gfCNCPoint1[26395] = {X 109.0469, Y 40.8285, Z -2.1667, A 0.000, B 0.000, C 0.000 }
gfCNCPoint1[26396] = {X 109.0468, Y 39.7004, Z -2.1667, A 0.000, B 0.000, C 0.000 }
gfCNCPoint1[26397] = {X 108.5557, Y 40.9005, Z -2.1667, A 0.000, B 0.000, C 0.000 }
gfCNCPoint1[26398] = {X 108.5557, Y 40.9005, Z 0.8333, A 0.000, B 0.000, C 0.000 }
gfCNCPoint1[26399] = {X 108.5557, Y 40.9005, Z 11.0000, A 0.000, B 0.000, C 0.000 }
gfCNCPoint1[26400] = {X 95.6842, Y 40.8760, Z 11.0000, A 0.000, B 0.000, C 0.000 }
gfCNCPoint1[26401] = {X 95.6842, Y 40.8760, Z 1.6667, A 0.000, B 0.000, C 0.000 }
gfCNCPoint1[26402] = {X 95.6842, Y 40.8760, Z -2.1667, A 0.000, B 0.000, C 0.000 }
gfCNCPoint1[26403] = {X 95.2101, Y 39.7165, Z -2.1667, A 0.000, B 0.000, C 0.000 }
gfCNCPoint1[26404] = {X 95.2102, Y 40.8690, Z -2.1667, A 0.000, B 0.000, C 0.000 }
gfCNCPoint1[26405] = {X 95.7335, Y 41.4123, Z -2.1667, A 0.000, B 0.000, C 0.000 }
gfCNCPoint1[26406] = {X 96.1583, Y 42.0355, Z -2.1667, A 0.000, B 0.000, C 0.000 }
gfCNCPoint1[26407] = {X 95.6842, Y 40.8760, Z -2.1667, A 0.000, B 0.000, C 0.000 }
gfCNCPoint1[26408] = {X 95.6842, Y 40.8760, Z 0.8333, A 0.000, B 0.000, C 0.000 }
gfCNCPoint1[26409] = {X 95.6842, Y 40.8760, Z 11.0000, A 0.000, B 0.000, C 0.000 }
gfCNCPoint1[26410] = {X -7.6965, Y 43.1560, Z 11.0000, A 0.000, B 0.000, C 0.000 }
gfCNCPoint1[26411] = {X -7.6965, Y 43.1560, Z 0.8333, A 0.000, B 0.000, C 0.000 }
gfCNCPoint1[26412] = {X -7.6965, Y 43.1560, Z -2.1667, A 0.000, B 0.000, C 0.000 }
gfCNCPoint1[26413] = {X -3.6965, Y 30.8015, Z -2.1667, A 0.000, B 0.000, C 0.000 }
gfCNCPoint1[26414] = {X -3.3664, Y 29.8871, Z -2.1667, A 0.000, B 0.000, C 0.000 }
gfCNCPoint1[26415] = {X -2.9760, Y 28.9968, Z -2.1667, A 0.000, B 0.000, C 0.000 }
gfCNCPoint1[26416] = {X -2.3495, Y 27.8703, Z -2.1667, A 0.000, B 0.000, C 0.000 }
gfCNCPoint1[26417] = {X -1.5931, Y 26.8265, Z -2.1667, A 0.000, B 0.000, C 0.000 }
gfCNCPoint1[26418] = {X -0.7177, Y 25.8802, Z -2.1667, A 0.000, B 0.000, C 0.000 }
gfCNCPoint1[26419] = {X 0.2642, Y 25.0451, Z -2.1667, A 0.000, B 0.000, C 0.000 }
gfCNCPoint1[26420] = {X 1.3386, Y 24.3329, Z -2.1667, A 0.000, B 0.000, C 0.000 }
gfCNCPoint1[26421] = {X 0.5787, Y 23.9225, Z -2.1667, A 0.000, B 0.000, C 0.000 }
gfCNCPoint1[26422] = {X -0.0865, Y 23.3717, Z -2.1667, A 0.000, B 0.000, C 0.000 }
gfCNCPoint1[26423] = {X -0.6312, Y 22.7015, Z -2.1667, A 0.000, B 0.000, C 0.000 }
gfCNCPoint1[26424] = {X -1.0345, Y 21.9378, Z -2.1667, A 0.000, B 0.000, C 0.000 }
gfCNCPoint1[26425] = {X -3.6458, Y 15.5423, Z -2.1667, A 0.000, B 0.000, C 0.000 }
gfCNCPoint1[26426] = {X -3.6716, Y 15.4775, Z -2.1667, A 0.000, B 0.000, C 0.000 }
gfCNCPoint1[26427] = {X -3.6965, Y 15.4122, Z -2.1667, A 0.000, B 0.000, C 0.000 }
gfCNCPoint1[26428] = {X -7.6965, Y 4.6517, Z -2.1667, A 0.000, B 0.000, C 0.000 }
gfCNCPoint1[26429] = {X -7.6965, Y 4.6517, Z 0.8333, A 0.000, B 0.000, C 0.000 }
gfCNCPoint1[26430] = {X -7.6965, Y 4.6517, Z 11.0000, A 0.000, B 0.000, C 0.000 }
gfCNCPoint1[26431] = {X -7.6965, Y 16.4123, Z 11.0000, A 0.000, B 0.000, C 0.000 }
gfCNCPoint1[26432] = {X -7.6965, Y 16.4123, Z 0.8333, A 0.000, B 0.000, C 0.000 }
gfCNCPoint1[26433] = {X -7.6965, Y 16.4123, Z -2.1667, A 0.000, B 0.000, C 0.000 }
gfCNCPoint1[26434] = {X -4.8869, Y 16.4123, Z -2.1667, A 0.000, B 0.000, C 0.000 }
gfCNCPoint1[26435] = {X -3.6965, Y 12.5935, Z -2.1667, A 0.000, B 0.000, C 0.000 }
gfCNCPoint1[26436] = {X -3.6605, Y 12.4832, Z -2.1667, A 0.000, B 0.000, C 0.000 }
gfCNCPoint1[26437] = {X -3.6215, Y 12.3739, Z -2.1667, A 0.000, B 0.000, C 0.000 }
gfCNCPoint1[26438] = {X -3.1666, Y 11.4827, Z -2.1667, A 0.000, B 0.000, C 0.000 }
gfCNCPoint1[26439] = {X -2.5188, Y 10.7200, Z -2.1667, A 0.000, B 0.000, C 0.000 }
gfCNCPoint1[26440] = {X -1.7129, Y 10.1268, Z -2.1667, A 0.000, B 0.000, C 0.000 }
gfCNCPoint1[26441] = {X -1.1157, Y 9.7861, Z -2.1667, A 0.000, B 0.000, C 0.000 }
gfCNCPoint1[26442] = {X -0.2291, Y 9.4045, Z -2.1667, A 0.000, B 0.000, C 0.000 }
gfCNCPoint1[26443] = {X 0.7202, Y 9.2292, Z -2.1667, A 0.000, B 0.000, C 0.000 }
gfCNCPoint1[26444] = {X 1.6847, Y 9.2691, Z -2.1667, A 0.000, B 0.000, C 0.000 }
gfCNCPoint1[26445] = {X 2.6162, Y 9.5222, Z -2.1667, A 0.000, B 0.000, C 0.000 }
gfCNCPoint1[26446] = {X 3.3958, Y 9.1594, Z -2.1667, A 0.000, B 0.000, C 0.000 }
gfCNCPoint1[26447] = {X 4.1961, Y 8.8448, Z -2.1667, A 0.000, B 0.000, C 0.000 }
gfCNCPoint1[26448] = {X 6.1070, Y 8.1762, Z -2.1667, A 0.000, B 0.000, C 0.000 }
gfCNCPoint1[26449] = {X 8.0685, Y 7.6747, Z -2.1667, A 0.000, B 0.000, C 0.000 }
gfCNCPoint1[26450] = {X 10.0658, Y 7.3442, Z -2.1667, A 0.000, B 0.000, C 0.000 }
gfCNCPoint1[26451] = {X 12.0843, Y 7.1871, Z -2.1667, A 0.000, B 0.000, C 0.000 }
gfCNCPoint1[26452] = {X 14.1088, Y 7.2045, Z -2.1667, A 0.000, B 0.000, C 0.000 }
gfCNCPoint1[26453] = {X 16.1242, Y 7.3964, Z -2.1667, A 0.000, B 0.000, C 0.000 }
gfCNCPoint1[26454] = {X 17.9474, Y 7.7301, Z -2.1667, A 0.000, B 0.000, C 0.000 }
gfCNCPoint1[26455] = {X 19.7250, Y 8.2552, Z -2.1667, A 0.000, B 0.000, C 0.000 }
gfCNCPoint1[26456] = {X 21.4368, Y 8.9658, Z -2.1667, A 0.000, B 0.000, C 0.000 }
gfCNCPoint1[26457] = {X 23.0637, Y 9.8538, Z -2.1667, A 0.000, B 0.000, C 0.000 }
gfCNCPoint1[26458] = {X 24.5873, Y 10.9093, Z -2.1667, A 0.000, B 0.000, C 0.000 }
gfCNCPoint1[26459] = {X 25.6719, Y 11.8584, Z -2.1667, A 0.000, B 0.000, C 0.000 }
gfCNCPoint1[26460] = {X 26.6450, Y 12.9216, Z -2.1667, A 0.000, B 0.000, C 0.000 }
gfCNCPoint1[26461] = {X 27.4945, Y 14.0858, Z -2.1667, A 0.000, B 0.000, C 0.000 }
gfCNCPoint1[26462] = {X 28.2102, Y 15.3368, Z -2.1667, A 0.000, B 0.000, C 0.000 }
gfCNCPoint1[26463] = {X 28.7831, Y 16.6592, Z -2.1667, A 0.000, B 0.000, C 0.000 }
gfCNCPoint1[26464] = {X 29.2588, Y 18.3155, Z -2.1667, A 0.000, B 0.000, C 0.000 }
gfCNCPoint1[26465] = {X 29.5409, Y 20.0155, Z -2.1667, A 0.000, B 0.000, C 0.000 }
gfCNCPoint1[26466] = {X 29.6260, Y 21.7366, Z -2.1667, A 0.000, B 0.000, C 0.000 }
gfCNCPoint1[26467] = {X 29.5127, Y 23.4561, Z -2.1667, A 0.000, B 0.000, C 0.000 }
gfCNCPoint1[26468] = {X 29.2026, Y 25.1512, Z -2.1667, A 0.000, B 0.000, C 0.000 }
gfCNCPoint1[26469] = {X 28.7606, Y 26.5973, Z -2.1667, A 0.000, B 0.000, C 0.000 }
gfCNCPoint1[26470] = {X 28.1355, Y 27.9743, Z -2.1667, A 0.000, B 0.000, C 0.000 }
gfCNCPoint1[26471] = {X 27.3378, Y 29.2590, Z -2.1667, A 0.000, B 0.000, C 0.000 }
gfCNCPoint1[26472] = {X 26.3810, Y 30.4299, Z -2.1667, A 0.000, B 0.000, C 0.000 }
gfCNCPoint1[26473] = {X 25.2809, Y 31.4676, Z -2.1667, A 0.000, B 0.000, C 0.000 }
gfCNCPoint1[26474] = {X 26.0850, Y 31.8097, Z -2.1667, A 0.000, B 0.000, C 0.000 }
gfCNCPoint1[26475] = {X 26.8038, Y 32.3066, Z -2.1667, A 0.000, B 0.000, C 0.000 }
gfCNCPoint1[26476] = {X 27.4079, Y 32.9381, Z -2.1667, A 0.000, B 0.000, C 0.000 }
gfCNCPoint1[26477] = {X 27.8726, Y 33.6781, Z -2.1667, A 0.000, B 0.000, C 0.000 }
gfCNCPoint1[26478] = {X 30.9100, Y 39.9530, Z -2.1667, A 0.000, B 0.000, C 0.000 }
gfCNCPoint1[26479] = {X 31.2306, Y 40.8622, Z -2.1667, A 0.000, B 0.000, C 0.000 }
gfCNCPoint1[26480] = {X 31.3415, Y 41.8197, Z -2.1667, A 0.000, B 0.000, C 0.000 }
gfCNCPoint1[26481] = {X 31.2374, Y 42.7781, Z -2.1667, A 0.000, B 0.000, C 0.000 }
gfCNCPoint1[26482] = {X 30.9234, Y 43.6895, Z -2.1667, A 0.000, B 0.000, C 0.000 }
gfCNCPoint1[26483] = {X 30.4150, Y 44.5085, Z -2.1667, A 0.000, B 0.000, C 0.000 }
gfCNCPoint1[26484] = {X 29.7377, Y 45.1945, Z -2.1667, A 0.000, B 0.000, C 0.000 }
gfCNCPoint1[26485] = {X 29.2014, Y 45.6281, Z -2.1667, A 0.000, B 0.000, C 0.000 }
gfCNCPoint1[26486] = {X 28.4966, Y 46.0912, Z -2.1667, A 0.000, B 0.000, C 0.000 }
gfCNCPoint1[26487] = {X 27.7155, Y 46.4091, Z -2.1667, A 0.000, B 0.000, C 0.000 }
gfCNCPoint1[26488] = {X 26.8877, Y 46.5699, Z -2.1667, A 0.000, B 0.000, C 0.000 }
gfCNCPoint1[26489] = {X 26.0445, Y 46.5675, Z -2.1667, A 0.000, B 0.000, C 0.000 }
gfCNCPoint1[26490] = {X 25.2176, Y 46.4020, Z -2.1667, A 0.000, B 0.000, C 0.000 }
gfCNCPoint1[26491] = {X 23.1996, Y 47.4597, Z -2.1667, A 0.000, B 0.000, C 0.000 }
gfCNCPoint1[26492] = {X 21.1036, Y 48.3530, Z -2.1667, A 0.000, B 0.000, C 0.000 }
gfCNCPoint1[26493] = {X 18.9430, Y 49.0760, Z -2.1667, A 0.000, B 0.000, C 0.000 }
gfCNCPoint1[26494] = {X 16.8434, Y 49.5947, Z -2.1667, A 0.000, B 0.000, C 0.000 }
gfCNCPoint1[26495] = {X 14.7038, Y 49.9107, Z -2.1667, A 0.000, B 0.000, C 0.000 }
gfCNCPoint1[26496] = {X 12.5438, Y 50.0209, Z -2.1667, A 0.000, B 0.000, C 0.000 }
gfCNCPoint1[26497] = {X 10.3832, Y 49.9245, Z -2.1667, A 0.000, B 0.000, C 0.000 }
gfCNCPoint1[26498] = {X 8.2417, Y 49.6223, Z -2.1667, A 0.000, B 0.000, C 0.000 }
gfCNCPoint1[26499] = {X 6.4092, Y 49.1801, Z -2.1667, A 0.000, B 0.000, C 0.000 }
gfCNCPoint1[26500] = {X 4.6364, Y 48.5391, Z -2.1667, A 0.000, B 0.000, C 0.000 }
gfCNCPoint1[26501] = {X 2.9448, Y 47.7071, Z -2.1667, A 0.000, B 0.000, C 0.000 }
gfCNCPoint1[26502] = {X 1.3550, Y 46.6941, Z -2.1667, A 0.000, B 0.000, C 0.000 }
gfCNCPoint1[26503] = {X 0.0296, Y 45.6271, Z -2.1667, A 0.000, B 0.000, C 0.000 }
gfCNCPoint1[26504] = {X -1.1487, Y 44.3994, Z -2.1667, A 0.000, B 0.000, C 0.000 }
gfCNCPoint1[26505] = {X -2.1603, Y 43.0312, Z -2.1667, A 0.000, B 0.000, C 0.000 }
gfCNCPoint1[26506] = {X -2.9888, Y 41.5449, Z -2.1667, A 0.000, B 0.000, C 0.000 }
gfCNCPoint1[26507] = {X -3.6205, Y 39.9650, Z -2.1667, A 0.000, B 0.000, C 0.000 }
gfCNCPoint1[26508] = {X -3.6590, Y 39.8451, Z -2.1667, A 0.000, B 0.000, C 0.000 }
gfCNCPoint1[26509] = {X -3.6965, Y 39.7249, Z -2.1667, A 0.000, B 0.000, C 0.000 }
gfCNCPoint1[26510] = {X -4.8683, Y 35.9004, Z -2.1667, A 0.000, B 0.000, C 0.000 }
gfCNCPoint1[26511] = {X -7.9903, Y 36.0269, Z -2.1667, A 0.000, B 0.000, C 0.000 }
gfCNCPoint1[26512] = {X -7.9903, Y 36.0269, Z 0.8333, A 0.000, B 0.000, C 0.000 }
gfCNCPoint1[26513] = {X -7.9903, Y 36.0269, Z 11.0000, A 0.000, B 0.000, C 0.000 }
gfCNCPoint1[26514] = {X 608.0000, Y 40.1203, Z 11.0000, A 0.000, B 0.000, C 0.000 }
gfCNCPoint1[26515] = {X 608.0000, Y 40.1203, Z 0.8333, A 0.000, B 0.000, C 0.000 }
gfCNCPoint1[26516] = {X 608.0000, Y 40.1203, Z -2.1667, A 0.000, B 0.000, C 0.000 }
gfCNCPoint1[26517] = {X 603.6965, Y 47.2357, Z -2.1667, A 0.000, B 0.000, C 0.000 }
gfCNCPoint1[26518] = {X 603.6633, Y 47.2897, Z -2.1667, A 0.000, B 0.000, C 0.000 }
gfCNCPoint1[26519] = {X 603.6293, Y 47.3432, Z -2.1667, A 0.000, B 0.000, C 0.000 }
gfCNCPoint1[26520] = {X 603.0929, Y 48.0160, Z -2.1667, A 0.000, B 0.000, C 0.000 }
gfCNCPoint1[26521] = {X 602.4339, Y 48.5691, Z -2.1667, A 0.000, B 0.000, C 0.000 }
gfCNCPoint1[26522] = {X 601.6783, Y 48.9807, Z -2.1667, A 0.000, B 0.000, C 0.000 }
gfCNCPoint1[26523] = {X 600.8561, Y 49.2343, Z -2.1667, A 0.000, B 0.000, C 0.000 }
gfCNCPoint1[26524] = {X 600.0000, Y 49.3200, Z -2.1667, A 0.000, B 0.000, C 0.000 }
gfCNCPoint1[26525] = {X 593.5565, Y 49.3200, Z -2.1667, A 0.000, B 0.000, C 0.000 }
gfCNCPoint1[26526] = {X 592.5952, Y 49.2117, Z -2.1667, A 0.000, B 0.000, C 0.000 }
gfCNCPoint1[26527] = {X 591.6822, Y 48.8922, Z -2.1667, A 0.000, B 0.000, C 0.000 }
gfCNCPoint1[26528] = {X 590.8631, Y 48.3775, Z -2.1667, A 0.000, B 0.000, C 0.000 }
gfCNCPoint1[26529] = {X 590.1790, Y 47.6935, Z -2.1667, A 0.000, B 0.000, C 0.000 }
gfCNCPoint1[26530] = {X 589.6643, Y 46.8744, Z -2.1667, A 0.000, B 0.000, C 0.000 }
gfCNCPoint1[26531] = {X 589.3448, Y 45.9613, Z -2.1667, A 0.000, B 0.000, C 0.000 }
gfCNCPoint1[26532] = {X 589.2365, Y 45.0000, Z -2.1667, A 0.000, B 0.000, C 0.000 }
gfCNCPoint1[26533] = {X 589.2365, Y 44.0643, Z -2.1667, A 0.000, B 0.000, C 0.000 }
gfCNCPoint1[26534] = {X 589.3414, Y 43.1363, Z -2.1667, A 0.000, B 0.000, C 0.000 }
gfCNCPoint1[26535] = {X 589.6413, Y 42.2518, Z -2.1667, A 0.000, B 0.000, C 0.000 }
gfCNCPoint1[26536] = {X 590.1226, Y 41.4513, Z -2.1667, A 0.000, B 0.000, C 0.000 }
gfCNCPoint1[26537] = {X 590.7631, Y 40.7716, Z -2.1667, A 0.000, B 0.000, C 0.000 }
gfCNCPoint1[26538] = {X 590.7634, Y 33.5293, Z -2.1667, A 0.000, B 0.000, C 0.000 }
gfCNCPoint1[26539] = {X 585.4453, Y 46.6524, Z -2.1667, A 0.000, B 0.000, C 0.000 }
gfCNCPoint1[26540] = {X 585.0755, Y 47.3550, Z -2.1667, A 0.000, B 0.000, C 0.000 }
gfCNCPoint1[26541] = {X 584.5834, Y 47.9780, Z -2.1667, A 0.000, B 0.000, C 0.000 }
gfCNCPoint1[26542] = {X 583.9856, Y 48.5004, Z -2.1667, A 0.000, B 0.000, C 0.000 }
gfCNCPoint1[26543] = {X 583.3023, Y 48.9046, Z -2.1667, A 0.000, B 0.000, C 0.000 }
gfCNCPoint1[26544] = {X 582.3585, Y 49.2242, Z -2.1667, A 0.000, B 0.000, C 0.000 }
gfCNCPoint1[26545] = {X 581.3666, Y 49.3191, Z -2.1667, A 0.000, B 0.000, C 0.000 }
gfCNCPoint1[26546] = {X 580.3794, Y 49.1842, Z -2.1667, A 0.000, B 0.000, C 0.000 }
gfCNCPoint1[26547] = {X 579.4493, Y 48.8268, Z -2.1667, A 0.000, B 0.000, C 0.000 }
gfCNCPoint1[26548] = {X 578.6259, Y 48.2657, Z -2.1667, A 0.000, B 0.000, C 0.000 }
gfCNCPoint1[26549] = {X 577.9529, Y 47.5309, Z -2.1667, A 0.000, B 0.000, C 0.000 }
gfCNCPoint1[26550] = {X 577.4662, Y 46.6615, Z -2.1667, A 0.000, B 0.000, C 0.000 }
gfCNCPoint1[26551] = {X 572.0179, Y 33.3391, Z -2.1667, A 0.000, B 0.000, C 0.000 }
gfCNCPoint1[26552] = {X 572.0183, Y 40.7709, Z -2.1667, A 0.000, B 0.000, C 0.000 }
gfCNCPoint1[26553] = {X 572.6568, Y 41.4417, Z -2.1667, A 0.000, B 0.000, C 0.000 }
gfCNCPoint1[26554] = {X 573.1376, Y 42.2332, Z -2.1667, A 0.000, B 0.000, C 0.000 }
gfCNCPoint1[26555] = {X 573.4387, Y 43.1089, Z -2.1667, A 0.000, B 0.000, C 0.000 }
gfCNCPoint1[26556] = {X 573.5463, Y 44.0287, Z -2.1667, A 0.000, B 0.000, C 0.000 }
gfCNCPoint1[26557] = {X 573.5464, Y 45.0000, Z -2.1667, A 0.000, B 0.000, C 0.000 }
gfCNCPoint1[26558] = {X 573.4381, Y 45.9613, Z -2.1667, A 0.000, B 0.000, C 0.000 }
gfCNCPoint1[26559] = {X 573.1186, Y 46.8744, Z -2.1667, A 0.000, B 0.000, C 0.000 }
gfCNCPoint1[26560] = {X 572.6039, Y 47.6935, Z -2.1667, A 0.000, B 0.000, C 0.000 }
gfCNCPoint1[26561] = {X 571.9199, Y 48.3775, Z -2.1667, A 0.000, B 0.000, C 0.000 }
gfCNCPoint1[26562] = {X 571.1008, Y 48.8922, Z -2.1667, A 0.000, B 0.000, C 0.000 }
gfCNCPoint1[26563] = {X 570.1877, Y 49.2117, Z -2.1667, A 0.000, B 0.000, C 0.000 }
gfCNCPoint1[26564] = {X 569.2264, Y 49.3200, Z -2.1667, A 0.000, B 0.000, C 0.000 }
gfCNCPoint1[26565] = {X 562.4443, Y 49.3200, Z -2.1667, A 0.000, B 0.000, C 0.000 }
gfCNCPoint1[26566] = {X 561.4830, Y 49.2117, Z -2.1667, A 0.000, B 0.000, C 0.000 }
gfCNCPoint1[26567] = {X 560.5699, Y 48.8922, Z -2.1667, A 0.000, B 0.000, C 0.000 }
gfCNCPoint1[26568] = {X 559.7508, Y 48.3775, Z -2.1667, A 0.000, B 0.000, C 0.000 }
gfCNCPoint1[26569] = {X 559.0668, Y 47.6935, Z -2.1667, A 0.000, B 0.000, C 0.000 }
gfCNCPoint1[26570] = {X 558.5521, Y 46.8744, Z -2.1667, A 0.000, B 0.000, C 0.000 }
gfCNCPoint1[26571] = {X 558.2326, Y 45.9613, Z -2.1667, A 0.000, B 0.000, C 0.000 }
gfCNCPoint1[26572] = {X 558.1243, Y 45.0000, Z -2.1667, A 0.000, B 0.000, C 0.000 }
gfCNCPoint1[26573] = {X 558.1243, Y 44.0645, Z -2.1667, A 0.000, B 0.000, C 0.000 }
gfCNCPoint1[26574] = {X 558.2290, Y 43.1360, Z -2.1667, A 0.000, B 0.000, C 0.000 }
gfCNCPoint1[26575] = {X 558.5292, Y 42.2511, Z -2.1667, A 0.000, B 0.000, C 0.000 }
gfCNCPoint1[26576] = {X 559.0111, Y 41.4507, Z -2.1667, A 0.000, B 0.000, C 0.000 }
gfCNCPoint1[26577] = {X 559.6527, Y 40.7713, Z -2.1667, A 0.000, B 0.000, C 0.000 }
gfCNCPoint1[26578] = {X 559.6527, Y 9.2309, Z -2.1667, A 0.000, B 0.000, C 0.000 }
gfCNCPoint1[26579] = {X 559.0139, Y 8.5599, Z -2.1667, A 0.000, B 0.000, C 0.000 }
gfCNCPoint1[26580] = {X 558.5330, Y 7.7681, Z -2.1667, A 0.000, B 0.000, C 0.000 }
gfCNCPoint1[26581] = {X 558.2318, Y 6.8920, Z -2.1667, A 0.000, B 0.000, C 0.000 }
gfCNCPoint1[26582] = {X 558.1245, Y 5.9718, Z -2.1667, A 0.000, B 0.000, C 0.000 }
gfCNCPoint1[26583] = {X 558.1243, Y 5.0000, Z -2.1667, A 0.000, B 0.000, C 0.000 }
gfCNCPoint1[26584] = {X 558.2326, Y 4.0387, Z -2.1667, A 0.000, B 0.000, C 0.000 }
gfCNCPoint1[26585] = {X 558.5521, Y 3.1256, Z -2.1667, A 0.000, B 0.000, C 0.000 }
gfCNCPoint1[26586] = {X 559.0668, Y 2.3065, Z -2.1667, A 0.000, B 0.000, C 0.000 }
gfCNCPoint1[26587] = {X 559.7508, Y 1.6225, Z -2.1667, A 0.000, B 0.000, C 0.000 }
gfCNCPoint1[26588] = {X 560.5699, Y 1.1078, Z -2.1667, A 0.000, B 0.000, C 0.000 }
gfCNCPoint1[26589] = {X 561.4830, Y 0.7883, Z -2.1667, A 0.000, B 0.000, C 0.000 }
gfCNCPoint1[26590] = {X 562.4443, Y 0.6800, Z -2.1667, A 0.000, B 0.000, C 0.000 }
gfCNCPoint1[26591] = {X 570.9376, Y 0.6800, Z -2.1667, A 0.000, B 0.000, C 0.000 }
gfCNCPoint1[26592] = {X 571.8988, Y 0.7883, Z -2.1667, A 0.000, B 0.000, C 0.000 }
gfCNCPoint1[26593] = {X 572.8119, Y 1.1078, Z -2.1667, A 0.000, B 0.000, C 0.000 }
gfCNCPoint1[26594] = {X 573.6310, Y 1.6225, Z -2.1667, A 0.000, B 0.000, C 0.000 }
gfCNCPoint1[26595] = {X 574.3151, Y 2.3065, Z -2.1667, A 0.000, B 0.000, C 0.000 }
gfCNCPoint1[26596] = {X 574.8297, Y 3.1256, Z -2.1667, A 0.000, B 0.000, C 0.000 }
gfCNCPoint1[26597] = {X 575.1492, Y 4.0387, Z -2.1667, A 0.000, B 0.000, C 0.000 }
gfCNCPoint1[26598] = {X 575.2576, Y 5.0000, Z -2.1667, A 0.000, B 0.000, C 0.000 }
gfCNCPoint1[26599] = {X 575.2576, Y 5.9342, Z -2.1667, A 0.000, B 0.000, C 0.000 }
gfCNCPoint1[26600] = {X 575.1862, Y 6.7158, Z -2.1667, A 0.000, B 0.000, C 0.000 }
gfCNCPoint1[26601] = {X 574.9747, Y 7.4715, Z -2.1667, A 0.000, B 0.000, C 0.000 }
gfCNCPoint1[26602] = {X 574.6299, Y 8.1766, Z -2.1667, A 0.000, B 0.000, C 0.000 }
gfCNCPoint1[26603] = {X 574.6075, Y 8.2193, Z -2.1667, A 0.000, B 0.000, C 0.000 }
gfCNCPoint1[26604] = {X 581.1909, Y 24.3708, Z -2.1667, A 0.000, B 0.000, C 0.000 }
gfCNCPoint1[26605] = {X 587.8460, Y 8.0945, Z -2.1667, A 0.000, B 0.000, C 0.000 }
gfCNCPoint1[26606] = {X 587.5318, Y 7.4233, Z -2.1667, A 0.000, B 0.000, C 0.000 }
gfCNCPoint1[26607] = {X 587.3369, Y 6.7083, Z -2.1667, A 0.000, B 0.000, C 0.000 }
gfCNCPoint1[26608] = {X 587.2671, Y 5.9705, Z -2.1667, A 0.000, B 0.000, C 0.000 }
gfCNCPoint1[26609] = {X 587.2670, Y 5.0000, Z -2.1667, A 0.000, B 0.000, C 0.000 }
gfCNCPoint1[26610] = {X 587.3753, Y 4.0387, Z -2.1667, A 0.000, B 0.000, C 0.000 }
gfCNCPoint1[26611] = {X 587.6948, Y 3.1256, Z -2.1667, A 0.000, B 0.000, C 0.000 }
gfCNCPoint1[26612] = {X 588.2094, Y 2.3065, Z -2.1667, A 0.000, B 0.000, C 0.000 }
gfCNCPoint1[26613] = {X 588.8935, Y 1.6225, Z -2.1667, A 0.000, B 0.000, C 0.000 }
gfCNCPoint1[26614] = {X 589.7126, Y 1.1078, Z -2.1667, A 0.000, B 0.000, C 0.000 }
gfCNCPoint1[26615] = {X 590.6257, Y 0.7883, Z -2.1667, A 0.000, B 0.000, C 0.000 }
gfCNCPoint1[26616] = {X 591.5870, Y 0.6800, Z -2.1667, A 0.000, B 0.000, C 0.000 }
gfCNCPoint1[26617] = {X 600.0000, Y 0.6800, Z -2.1667, A 0.000, B 0.000, C 0.000 }
gfCNCPoint1[26618] = {X 600.8561, Y 0.7657, Z -2.1667, A 0.000, B 0.000, C 0.000 }
gfCNCPoint1[26619] = {X 601.6783, Y 1.0193, Z -2.1667, A 0.000, B 0.000, C 0.000 }
gfCNCPoint1[26620] = {X 602.4339, Y 1.4309, Z -2.1667, A 0.000, B 0.000, C 0.000 }
gfCNCPoint1[26621] = {X 603.0929, Y 1.9840, Z -2.1667, A 0.000, B 0.000, C 0.000 }
gfCNCPoint1[26622] = {X 603.6293, Y 2.6568, Z -2.1667, A 0.000, B 0.000, C 0.000 }
gfCNCPoint1[26623] = {X 603.6633, Y 2.7103, Z -2.1667, A 0.000, B 0.000, C 0.000 }
gfCNCPoint1[26624] = {X 603.6965, Y 2.7643, Z -2.1667, A 0.000, B 0.000, C 0.000 }
gfCNCPoint1[26625] = {X 608.0000, Y 9.8797, Z -2.1667, A 0.000, B 0.000, C 0.000 }
gfCNCPoint1[26626] = {X 608.0000, Y 9.8797, Z 0.8333, A 0.000, B 0.000, C 0.000 }
gfCNCPoint1[26627] = {X 608.0000, Y 9.8797, Z 11.0000, A 0.000, B 0.000, C 0.000 }
gfCNCPoint1[26628] = {X -7.6965, Y 16.7861, Z 11.0000, A 0.000, B 0.000, C 0.000 }
gfCNCPoint1[26629] = {X -7.6965, Y 16.7861, Z 0.8333, A 0.000, B 0.000, C 0.000 }
gfCNCPoint1[26630] = {X -7.6965, Y 16.7861, Z -2.1667, A 0.000, B 0.000, C 0.000 }
gfCNCPoint1[26631] = {X -4.6247, Y 16.7861, Z -2.1667, A 0.000, B 0.000, C 0.000 }
gfCNCPoint1[26632] = {X -3.6965, Y 12.8952, Z -2.1667, A 0.000, B 0.000, C 0.000 }
gfCNCPoint1[26633] = {X -3.6290, Y 12.6462, Z -2.1667, A 0.000, B 0.000, C 0.000 }
gfCNCPoint1[26634] = {X -3.5465, Y 12.4018, Z -2.1667, A 0.000, B 0.000, C 0.000 }
gfCNCPoint1[26635] = {X -3.1000, Y 11.5270, Z -2.1667, A 0.000, B 0.000, C 0.000 }
gfCNCPoint1[26636] = {X -2.4642, Y 10.7785, Z -2.1667, A 0.000, B 0.000, C 0.000 }
gfCNCPoint1[26637] = {X -1.6733, Y 10.1963, Z -2.1667, A 0.000, B 0.000, C 0.000 }
gfCNCPoint1[26638] = {X -1.0761, Y 9.8556, Z -2.1667, A 0.000, B 0.000, C 0.000 }
gfCNCPoint1[26639] = {X -0.1973, Y 9.4784, Z -2.1667, A 0.000, B 0.000, C 0.000 }
gfCNCPoint1[26640] = {X 0.7437, Y 9.3078, Z -2.1667, A 0.000, B 0.000, C 0.000 }
gfCNCPoint1[26641] = {X 1.6990, Y 9.3524, Z -2.1667, A 0.000, B 0.000, C 0.000 }
gfCNCPoint1[26642] = {X 2.6199, Y 9.6099, Z -2.1667, A 0.000, B 0.000, C 0.000 }
gfCNCPoint1[26643] = {X 3.4114, Y 9.2397, Z -2.1667, A 0.000, B 0.000, C 0.000 }
gfCNCPoint1[26644] = {X 4.2244, Y 8.9197, Z -2.1667, A 0.000, B 0.000, C 0.000 }
gfCNCPoint1[26645] = {X 6.1291, Y 8.2531, Z -2.1667, A 0.000, B 0.000, C 0.000 }
gfCNCPoint1[26646] = {X 8.0841, Y 7.7532, Z -2.1667, A 0.000, B 0.000, C 0.000 }
gfCNCPoint1[26647] = {X 10.0750, Y 7.4237, Z -2.1667, A 0.000, B 0.000, C 0.000 }
gfCNCPoint1[26648] = {X 12.0868, Y 7.2671, Z -2.1667, A 0.000, B 0.000, C 0.000 }
gfCNCPoint1[26649] = {X 14.1047, Y 7.2844, Z -2.1667, A 0.000, B 0.000, C 0.000 }
gfCNCPoint1[26650] = {X 16.1136, Y 7.4757, Z -2.1667, A 0.000, B 0.000, C 0.000 }
gfCNCPoint1[26651] = {X 17.9285, Y 7.8078, Z -2.1667, A 0.000, B 0.000, C 0.000 }
gfCNCPoint1[26652] = {X 19.6980, Y 8.3305, Z -2.1667, A 0.000, B 0.000, C 0.000 }
gfCNCPoint1[26653] = {X 21.4021, Y 9.0378, Z -2.1667, A 0.000, B 0.000, C 0.000 }
gfCNCPoint1[26654] = {X 23.0217, Y 9.9218, Z -2.1667, A 0.000, B 0.000, C 0.000 }
gfCNCPoint1[26655] = {X 24.5383, Y 10.9726, Z -2.1667, A 0.000, B 0.000, C 0.000 }
gfCNCPoint1[26656] = {X 25.6162, Y 11.9158, Z -2.1667, A 0.000, B 0.000, C 0.000 }
gfCNCPoint1[26657] = {X 26.5832, Y 12.9724, Z -2.1667, A 0.000, B 0.000, C 0.000 }
gfCNCPoint1[26658] = {X 27.4275, Y 14.1294, Z -2.1667, A 0.000, B 0.000, C 0.000 }
gfCNCPoint1[26659] = {X 28.1387, Y 15.3726, Z -2.1667, A 0.000, B 0.000, C 0.000 }
gfCNCPoint1[26660] = {X 28.7081, Y 16.6869, Z -2.1667, A 0.000, B 0.000, C 0.000 }
gfCNCPoint1[26661] = {X 29.1810, Y 18.3342, Z -2.1667, A 0.000, B 0.000, C 0.000 }
gfCNCPoint1[26662] = {X 29.4615, Y 20.0249, Z -2.1667, A 0.000, B 0.000, C 0.000 }
gfCNCPoint1[26663] = {X 29.5460, Y 21.7366, Z -2.1667, A 0.000, B 0.000, C 0.000 }
gfCNCPoint1[26664] = {X 29.4332, Y 23.4467, Z -2.1667, A 0.000, B 0.000, C 0.000 }
gfCNCPoint1[26665] = {X 29.1248, Y 25.1325, Z -2.1667, A 0.000, B 0.000, C 0.000 }
gfCNCPoint1[26666] = {X 28.6750, Y 26.5972, Z -2.1667, A 0.000, B 0.000, C 0.000 }
gfCNCPoint1[26667] = {X 28.0363, Y 27.9898, Z -2.1667, A 0.000, B 0.000, C 0.000 }
gfCNCPoint1[26668] = {X 27.2196, Y 29.2862, Z -2.1667, A 0.000, B 0.000, C 0.000 }
gfCNCPoint1[26669] = {X 26.2393, Y 30.4637, Z -2.1667, A 0.000, B 0.000, C 0.000 }
gfCNCPoint1[26670] = {X 25.1125, Y 31.5019, Z -2.1667, A 0.000, B 0.000, C 0.000 }
gfCNCPoint1[26671] = {X 25.2520, Y 31.5424, Z -2.1667, A 0.000, B 0.000, C 0.000 }
gfCNCPoint1[26672] = {X 25.3901, Y 31.5876, Z -2.1667, A 0.000, B 0.000, C 0.000 }
gfCNCPoint1[26673] = {X 26.1377, Y 31.9315, Z -2.1667, A 0.000, B 0.000, C 0.000 }
gfCNCPoint1[26674] = {X 26.8048, Y 32.4133, Z -2.1667, A 0.000, B 0.000, C 0.000 }
gfCNCPoint1[26675] = {X 27.3662, Y 33.0149, Z -2.1667, A 0.000, B 0.000, C 0.000 }
gfCNCPoint1[26676] = {X 27.8009, Y 33.7136, Z -2.1667, A 0.000, B 0.000, C 0.000 }
gfCNCPoint1[26677] = {X 30.8380, Y 39.9879, Z -2.1667, A 0.000, B 0.000, C 0.000 }
gfCNCPoint1[26678] = {X 31.1526, Y 40.8802, Z -2.1667, A 0.000, B 0.000, C 0.000 }
gfCNCPoint1[26679] = {X 31.2615, Y 41.8200, Z -2.1667, A 0.000, B 0.000, C 0.000 }
gfCNCPoint1[26680] = {X 31.1593, Y 42.7606, Z -2.1667, A 0.000, B 0.000, C 0.000 }
gfCNCPoint1[26681] = {X 30.8511, Y 43.6551, Z -2.1667, A 0.000, B 0.000, C 0.000 }
gfCNCPoint1[26682] = {X 30.3522, Y 44.4590, Z -2.1667, A 0.000, B 0.000, C 0.000 }
gfCNCPoint1[26683] = {X 29.6874, Y 45.1323, Z -2.1667, A 0.000, B 0.000, C 0.000 }
gfCNCPoint1[26684] = {X 29.1511, Y 45.5659, Z -2.1667, A 0.000, B 0.000, C 0.000 }
gfCNCPoint1[26685] = {X 28.4532, Y 46.0236, Z -2.1667, A 0.000, B 0.000, C 0.000 }
gfCNCPoint1[26686] = {X 27.6795, Y 46.3363, Z -2.1667, A 0.000, B 0.000, C 0.000 }
gfCNCPoint1[26687] = {X 26.8595, Y 46.4922, Z -2.1667, A 0.000, B 0.000, C 0.000 }
gfCNCPoint1[26688] = {X 26.0250, Y 46.4850, Z -2.1667, A 0.000, B 0.000, C 0.000 }
gfCNCPoint1[26689] = {X 25.2078, Y 46.3153, Z -2.1667, A 0.000, B 0.000, C 0.000 }
gfCNCPoint1[26690] = {X 23.1862, Y 47.3775, Z -2.1667, A 0.000, B 0.000, C 0.000 }
gfCNCPoint1[26691] = {X 21.0859, Y 48.2741, Z -2.1667, A 0.000, B 0.000, C 0.000 }
gfCNCPoint1[26692] = {X 18.9204, Y 48.9993, Z -2.1667, A 0.000, B 0.000, C 0.000 }
gfCNCPoint1[26693] = {X 16.8281, Y 49.5162, Z -2.1667, A 0.000, B 0.000, C 0.000 }
gfCNCPoint1[26694] = {X 14.6960, Y 49.8311, Z -2.1667, A 0.000, B 0.000, C 0.000 }
gfCNCPoint1[26695] = {X 12.5436, Y 49.9409, Z -2.1667, A 0.000, B 0.000, C 0.000 }
gfCNCPoint1[26696] = {X 10.3905, Y 49.8448, Z -2.1667, A 0.000, B 0.000, C 0.000 }
gfCNCPoint1[26697] = {X 8.2564, Y 49.5436, Z -2.1667, A 0.000, B 0.000, C 0.000 }
gfCNCPoint1[26698] = {X 6.4323, Y 49.1035, Z -2.1667, A 0.000, B 0.000, C 0.000 }
gfCNCPoint1[26699] = {X 4.6677, Y 48.4655, Z -2.1667, A 0.000, B 0.000, C 0.000 }
gfCNCPoint1[26700] = {X 2.9839, Y 47.6373, Z -2.1667, A 0.000, B 0.000, C 0.000 }
gfCNCPoint1[26701] = {X 1.4014, Y 46.6289, Z -2.1667, A 0.000, B 0.000, C 0.000 }
gfCNCPoint1[26702] = {X 0.0838, Y 45.5683, Z -2.1667, A 0.000, B 0.000, C 0.000 }
gfCNCPoint1[26703] = {X -1.0874, Y 44.3480, Z -2.1667, A 0.000, B 0.000, C 0.000 }
gfCNCPoint1[26704] = {X -2.0930, Y 42.9880, Z -2.1667, A 0.000, B 0.000, C 0.000 }
gfCNCPoint1[26705] = {X -2.9165, Y 41.5106, Z -2.1667, A 0.000, B 0.000, C 0.000 }
gfCNCPoint1[26706] = {X -3.5444, Y 39.9401, Z -2.1667, A 0.000, B 0.000, C 0.000 }
gfCNCPoint1[26707] = {X -3.6229, Y 39.6920, Z -2.1667, A 0.000, B 0.000, C 0.000 }
gfCNCPoint1[26708] = {X -3.6965, Y 39.4424, Z -2.1667, A 0.000, B 0.000, C 0.000 }
gfCNCPoint1[26709] = {X -4.7898, Y 35.5948, Z -2.1667, A 0.000, B 0.000, C 0.000 }
gfCNCPoint1[26710] = {X -8.0015, Y 35.6599, Z -2.1667, A 0.000, B 0.000, C 0.000 }
gfCNCPoint1[26711] = {X -8.0015, Y 35.6599, Z 0.8333, A 0.000, B 0.000, C 0.000 }
gfCNCPoint1[26712] = {X -8.0015, Y 35.6599, Z 11.0000, A 0.000, B 0.000, C 0.000 }
gfCNCPoint1[26713] = {X -7.6965, Y 17.3007, Z 11.0000, A 0.000, B 0.000, C 0.000 }
gfCNCPoint1[26714] = {X -7.6965, Y 17.3007, Z 0.8333, A 0.000, B 0.000, C 0.000 }
gfCNCPoint1[26715] = {X -7.6965, Y 17.3007, Z -2.1667, A 0.000, B 0.000, C 0.000 }
gfCNCPoint1[26716] = {X -4.2196, Y 17.3007, Z -2.1667, A 0.000, B 0.000, C 0.000 }
gfCNCPoint1[26717] = {X -3.6965, Y 13.3350, Z -2.1667, A 0.000, B 0.000, C 0.000 }
gfCNCPoint1[26718] = {X -3.6095, Y 12.8760, Z -2.1667, A 0.000, B 0.000, C 0.000 }
gfCNCPoint1[26719] = {X -3.4715, Y 12.4296, Z -2.1667, A 0.000, B 0.000, C 0.000 }
gfCNCPoint1[26720] = {X -3.0334, Y 11.5714, Z -2.1667, A 0.000, B 0.000, C 0.000 }
gfCNCPoint1[26721] = {X -2.4097, Y 10.8370, Z -2.1667, A 0.000, B 0.000, C 0.000 }
gfCNCPoint1[26722] = {X -1.6337, Y 10.2658, Z -2.1667, A 0.000, B 0.000, C 0.000 }
gfCNCPoint1[26723] = {X -1.0364, Y 9.9251, Z -2.1667, A 0.000, B 0.000, C 0.000 }
gfCNCPoint1[26724] = {X -0.1655, Y 9.5524, Z -2.1667, A 0.000, B 0.000, C 0.000 }
gfCNCPoint1[26725] = {X 0.7671, Y 9.3865, Z -2.1667, A 0.000, B 0.000, C 0.000 }
gfCNCPoint1[26726] = {X 1.7131, Y 9.4358, Z -2.1667, A 0.000, B 0.000, C 0.000 }
gfCNCPoint1[26727] = {X 2.6235, Y 9.6979, Z -2.1667, A 0.000, B 0.000, C 0.000 }
gfCNCPoint1[26728] = {X 3.4269, Y 9.3202, Z -2.1667, A 0.000, B 0.000, C 0.000 }
gfCNCPoint1[26729] = {X 4.2527, Y 8.9945, Z -2.1667, A 0.000, B 0.000, C 0.000 }
gfCNCPoint1[26730] = {X 6.1511, Y 8.3300, Z -2.1667, A 0.000, B 0.000, C 0.000 }
gfCNCPoint1[26731] = {X 8.0997, Y 7.8317, Z -2.1667, A 0.000, B 0.000, C 0.000 }
gfCNCPoint1[26732] = {X 10.0841, Y 7.5032, Z -2.1667, A 0.000, B 0.000, C 0.000 }
gfCNCPoint1[26733] = {X 12.0894, Y 7.3470, Z -2.1667, A 0.000, B 0.000, C 0.000 }
gfCNCPoint1[26734] = {X 14.1006, Y 7.3643, Z -2.1667, A 0.000, B 0.000, C 0.000 }
gfCNCPoint1[26735] = {X 16.1029, Y 7.5550, Z -2.1667, A 0.000, B 0.000, C 0.000 }
gfCNCPoint1[26736] = {X 17.9096, Y 7.8856, Z -2.1667, A 0.000, B 0.000, C 0.000 }
gfCNCPoint1[26737] = {X 19.6711, Y 8.4058, Z -2.1667, A 0.000, B 0.000, C 0.000 }
gfCNCPoint1[26738] = {X 21.3674, Y 9.1099, Z -2.1667, A 0.000, B 0.000, C 0.000 }
gfCNCPoint1[26739] = {X 22.9796, Y 9.9899, Z -2.1667, A 0.000, B 0.000, C 0.000 }
gfCNCPoint1[26740] = {X 24.4894, Y 11.0358, Z -2.1667, A 0.000, B 0.000, C 0.000 }
gfCNCPoint1[26741] = {X 25.5605, Y 11.9732, Z -2.1667, A 0.000, B 0.000, C 0.000 }
gfCNCPoint1[26742] = {X 26.5214, Y 13.0232, Z -2.1667, A 0.000, B 0.000, C 0.000 }
gfCNCPoint1[26743] = {X 27.3604, Y 14.1730, Z -2.1667, A 0.000, B 0.000, C 0.000 }
gfCNCPoint1[26744] = {X 28.0672, Y 15.4085, Z -2.1667, A 0.000, B 0.000, C 0.000 }
gfCNCPoint1[26745] = {X 28.6330, Y 16.7146, Z -2.1667, A 0.000, B 0.000, C 0.000 }
gfCNCPoint1[26746] = {X 29.1032, Y 18.3529, Z -2.1667, A 0.000, B 0.000, C 0.000 }
gfCNCPoint1[26747] = {X 29.3821, Y 20.0343, Z -2.1667, A 0.000, B 0.000, C 0.000 }
gfCNCPoint1[26748] = {X 29.4660, Y 21.7366, Z -2.1667, A 0.000, B 0.000, C 0.000 }
gfCNCPoint1[26749] = {X 29.3538, Y 23.4373, Z -2.1667, A 0.000, B 0.000, C 0.000 }
gfCNCPoint1[26750] = {X 29.0470, Y 25.1139, Z -2.1667, A 0.000, B 0.000, C 0.000 }
gfCNCPoint1[26751] = {X 28.5888, Y 26.5986, Z -2.1667, A 0.000, B 0.000, C 0.000 }
gfCNCPoint1[26752] = {X 27.9351, Y 28.0083, Z -2.1667, A 0.000, B 0.000, C 0.000 }
gfCNCPoint1[26753] = {X 27.0977, Y 29.3172, Z -2.1667, A 0.000, B 0.000, C 0.000 }
gfCNCPoint1[26754] = {X 26.0919, Y 30.5016, Z -2.1667, A 0.000, B 0.000, C 0.000 }
gfCNCPoint1[26755] = {X 24.9359, Y 31.5400, Z -2.1667, A 0.000, B 0.000, C 0.000 }
gfCNCPoint1[26756] = {X 25.1516, Y 31.5959, Z -2.1667, A 0.000, B 0.000, C 0.000 }
gfCNCPoint1[26757] = {X 25.3639, Y 31.6632, Z -2.1667, A 0.000, B 0.000, C 0.000 }
gfCNCPoint1[26758] = {X 26.0974, Y 32.0006, Z -2.1667, A 0.000, B 0.000, C 0.000 }
gfCNCPoint1[26759] = {X 26.7518, Y 32.4733, Z -2.1667, A 0.000, B 0.000, C 0.000 }
gfCNCPoint1[26760] = {X 27.3027, Y 33.0635, Z -2.1667, A 0.000, B 0.000, C 0.000 }
gfCNCPoint1[26761] = {X 27.7292, Y 33.7491, Z -2.1667, A 0.000, B 0.000, C 0.000 }
gfCNCPoint1[26762] = {X 30.7660, Y 40.0227, Z -2.1667, A 0.000, B 0.000, C 0.000 }
gfCNCPoint1[26763] = {X 31.0747, Y 40.8982, Z -2.1667, A 0.000, B 0.000, C 0.000 }
gfCNCPoint1[26764] = {X 31.1815, Y 41.8203, Z -2.1667, A 0.000, B 0.000, C 0.000 }
gfCNCPoint1[26765] = {X 31.0813, Y 42.7431, Z -2.1667, A 0.000, B 0.000, C 0.000 }
gfCNCPoint1[26766] = {X 30.7789, Y 43.6208, Z -2.1667, A 0.000, B 0.000, C 0.000 }
gfCNCPoint1[26767] = {X 30.2893, Y 44.4095, Z -2.1667, A 0.000, B 0.000, C 0.000 }
gfCNCPoint1[26768] = {X 29.6371, Y 45.0700, Z -2.1667, A 0.000, B 0.000, C 0.000 }
gfCNCPoint1[26769] = {X 29.1009, Y 45.5036, Z -2.1667, A 0.000, B 0.000, C 0.000 }
gfCNCPoint1[26770] = {X 28.4099, Y 45.9559, Z -2.1667, A 0.000, B 0.000, C 0.000 }
gfCNCPoint1[26771] = {X 27.6435, Y 46.2635, Z -2.1667, A 0.000, B 0.000, C 0.000 }
gfCNCPoint1[26772] = {X 26.8314, Y 46.4143, Z -2.1667, A 0.000, B 0.000, C 0.000 }
gfCNCPoint1[26773] = {X 26.0056, Y 46.4024, Z -2.1667, A 0.000, B 0.000, C 0.000 }
gfCNCPoint1[26774] = {X 25.1983, Y 46.2283, Z -2.1667, A 0.000, B 0.000, C 0.000 }
gfCNCPoint1[26775] = {X 23.1730, Y 47.2952, Z -2.1667, A 0.000, B 0.000, C 0.000 }
gfCNCPoint1[26776] = {X 21.0683, Y 48.1952, Z -2.1667, A 0.000, B 0.000, C 0.000 }
gfCNCPoint1[26777] = {X 18.8978, Y 48.9225, Z -2.1667, A 0.000, B 0.000, C 0.000 }
gfCNCPoint1[26778] = {X 16.8128, Y 49.4377, Z -2.1667, A 0.000, B 0.000, C 0.000 }
gfCNCPoint1[26779] = {X 14.6882, Y 49.7514, Z -2.1667, A 0.000, B 0.000, C 0.000 }
gfCNCPoint1[26780] = {X 12.5433, Y 49.8609, Z -2.1667, A 0.000, B 0.000, C 0.000 }
gfCNCPoint1[26781] = {X 10.3977, Y 49.7652, Z -2.1667, A 0.000, B 0.000, C 0.000 }
gfCNCPoint1[26782] = {X 8.2711, Y 49.4650, Z -2.1667, A 0.000, B 0.000, C 0.000 }
gfCNCPoint1[26783] = {X 6.4554, Y 49.0270, Z -2.1667, A 0.000, B 0.000, C 0.000 }
gfCNCPoint1[26784] = {X 4.6989, Y 48.3919, Z -2.1667, A 0.000, B 0.000, C 0.000 }
gfCNCPoint1[26785] = {X 3.0230, Y 47.5675, Z -2.1667, A 0.000, B 0.000, C 0.000 }
gfCNCPoint1[26786] = {X 1.4478, Y 46.5637, Z -2.1667, A 0.000, B 0.000, C 0.000 }
gfCNCPoint1[26787] = {X 0.1381, Y 45.5096, Z -2.1667, A 0.000, B 0.000, C 0.000 }
gfCNCPoint1[26788] = {X -1.0261, Y 44.2966, Z -2.1667, A 0.000, B 0.000, C 0.000 }
gfCNCPoint1[26789] = {X -2.0256, Y 42.9448, Z -2.1667, A 0.000, B 0.000, C 0.000 }
gfCNCPoint1[26790] = {X -2.8442, Y 41.4763, Z -2.1667, A 0.000, B 0.000, C 0.000 }
gfCNCPoint1[26791] = {X -3.4684, Y 39.9152, Z -2.1667, A 0.000, B 0.000, C 0.000 }
gfCNCPoint1[26792] = {X -3.5884, Y 39.5283, Z -2.1667, A 0.000, B 0.000, C 0.000 }
gfCNCPoint1[26793] = {X -3.6965, Y 39.1378, Z -2.1667, A 0.000, B 0.000, C 0.000 }
gfCNCPoint1[26794] = {X -4.7036, Y 35.2667, Z -2.1667, A 0.000, B 0.000, C 0.000 }
gfCNCPoint1[26795] = {X -8.0052, Y 35.2612, Z -2.1667, A 0.000, B 0.000, C 0.000 }
gfCNCPoint1[26796] = {X -8.0052, Y 35.2612, Z 0.8333, A 0.000, B 0.000, C 0.000 }
gfCNCPoint1[26797] = {X -8.0052, Y 35.2612, Z 11.0000, A 0.000, B 0.000, C 0.000 }
gfCNCPoint1[26798] = {X -7.9989, Y 34.8122, Z 11.0000, A 0.000, B 0.000, C 0.000 }
gfCNCPoint1[26799] = {X -7.9989, Y 34.8122, Z 0.8333, A 0.000, B 0.000, C 0.000 }
gfCNCPoint1[26800] = {X -7.9989, Y 34.8122, Z -2.1667, A 0.000, B 0.000, C 0.000 }
gfCNCPoint1[26801] = {X -4.8617, Y 34.8949, Z -2.1667, A 0.000, B 0.000, C 0.000 }
gfCNCPoint1[26802] = {X -3.6965, Y 31.0684, Z -2.1667, A 0.000, B 0.000, C 0.000 }
gfCNCPoint1[26803] = {X -3.6590, Y 30.9471, Z -2.1667, A 0.000, B 0.000, C 0.000 }
gfCNCPoint1[26804] = {X -3.6204, Y 30.8261, Z -2.1667, A 0.000, B 0.000, C 0.000 }
gfCNCPoint1[26805] = {X -3.2922, Y 29.9170, Z -2.1667, A 0.000, B 0.000, C 0.000 }
gfCNCPoint1[26806] = {X -2.9041, Y 29.0318, Z -2.1667, A 0.000, B 0.000, C 0.000 }
gfCNCPoint1[26807] = {X -2.2643, Y 27.8856, Z -2.1667, A 0.000, B 0.000, C 0.000 }
gfCNCPoint1[26808] = {X -1.4892, Y 26.8262, Z -2.1667, A 0.000, B 0.000, C 0.000 }
gfCNCPoint1[26809] = {X -0.5903, Y 25.8695, Z -2.1667, A 0.000, B 0.000, C 0.000 }
gfCNCPoint1[26810] = {X 0.4188, Y 25.0299, Z -2.1667, A 0.000, B 0.000, C 0.000 }
gfCNCPoint1[26811] = {X 1.5229, Y 24.3199, Z -2.1667, A 0.000, B 0.000, C 0.000 }
gfCNCPoint1[26812] = {X 0.7350, Y 23.9290, Z -2.1667, A 0.000, B 0.000, C 0.000 }
gfCNCPoint1[26813] = {X 0.0426, Y 23.3866, Z -2.1667, A 0.000, B 0.000, C 0.000 }
gfCNCPoint1[26814] = {X -0.5256, Y 22.7152, Z -2.1667, A 0.000, B 0.000, C 0.000 }
gfCNCPoint1[26815] = {X -0.9460, Y 21.9427, Z -2.1667, A 0.000, B 0.000, C 0.000 }
gfCNCPoint1[26816] = {X -3.6215, Y 15.3844, Z -2.1667, A 0.000, B 0.000, C 0.000 }
gfCNCPoint1[26817] = {X -3.6605, Y 15.2751, Z -2.1667, A 0.000, B 0.000, C 0.000 }
gfCNCPoint1[26818] = {X -3.6965, Y 15.1647, Z -2.1667, A 0.000, B 0.000, C 0.000 }
gfCNCPoint1[26819] = {X -4.8869, Y 11.3460, Z -2.1667, A 0.000, B 0.000, C 0.000 }
gfCNCPoint1[26820] = {X -7.6965, Y 11.3460, Z -2.1667, A 0.000, B 0.000, C 0.000 }
gfCNCPoint1[26821] = {X -7.6965, Y 11.3460, Z 0.8333, A 0.000, B 0.000, C 0.000 }
gfCNCPoint1[26822] = {X -7.6965, Y 11.3460, Z 11.0000, A 0.000, B 0.000, C 0.000 }
gfCNCPoint1[26823] = {X -8.0049, Y 35.1798, Z 11.0000, A 0.000, B 0.000, C 0.000 }
gfCNCPoint1[26824] = {X -8.0049, Y 35.1798, Z 0.8333, A 0.000, B 0.000, C 0.000 }
gfCNCPoint1[26825] = {X -8.0049, Y 35.1798, Z -2.1667, A 0.000, B 0.000, C 0.000 }
gfCNCPoint1[26826] = {X -4.7896, Y 35.1995, Z -2.1667, A 0.000, B 0.000, C 0.000 }
gfCNCPoint1[26827] = {X -3.6965, Y 31.3518, Z -2.1667, A 0.000, B 0.000, C 0.000 }
gfCNCPoint1[26828] = {X -3.6226, Y 31.1006, Z -2.1667, A 0.000, B 0.000, C 0.000 }
gfCNCPoint1[26829] = {X -3.5443, Y 30.8508, Z -2.1667, A 0.000, B 0.000, C 0.000 }
gfCNCPoint1[26830] = {X -3.2179, Y 29.9467, Z -2.1667, A 0.000, B 0.000, C 0.000 }
gfCNCPoint1[26831] = {X -2.8320, Y 29.0664, Z -2.1667, A 0.000, B 0.000, C 0.000 }
gfCNCPoint1[26832] = {X -2.0400, Y 27.6912, Z -2.1667, A 0.000, B 0.000, C 0.000 }
gfCNCPoint1[26833] = {X -1.0522, Y 26.4491, Z -2.1667, A 0.000, B 0.000, C 0.000 }
gfCNCPoint1[26834] = {X 0.1094, Y 25.3677, Z -2.1667, A 0.000, B 0.000, C 0.000 }
gfCNCPoint1[26835] = {X 1.4189, Y 24.4713, Z -2.1667, A 0.000, B 0.000, C 0.000 }
gfCNCPoint1[26836] = {X 1.5680, Y 24.3864, Z -2.1667, A 0.000, B 0.000, C 0.000 }
gfCNCPoint1[26837] = {X 1.7185, Y 24.3039, Z -2.1667, A 0.000, B 0.000, C 0.000 }
gfCNCPoint1[26838] = {X 0.8915, Y 23.9306, Z -2.1667, A 0.000, B 0.000, C 0.000 }
gfCNCPoint1[26839] = {X 0.1627, Y 23.3899, Z -2.1667, A 0.000, B 0.000, C 0.000 }
gfCNCPoint1[26840] = {X -0.4343, Y 22.7066, Z -2.1667, A 0.000, B 0.000, C 0.000 }
gfCNCPoint1[26841] = {X -0.8722, Y 21.9118, Z -2.1667, A 0.000, B 0.000, C 0.000 }
gfCNCPoint1[26842] = {X -3.5465, Y 15.3565, Z -2.1667, A 0.000, B 0.000, C 0.000 }
gfCNCPoint1[26843] = {X -3.6290, Y 15.1120, Z -2.1667, A 0.000, B 0.000, C 0.000 }
gfCNCPoint1[26844] = {X -3.6965, Y 14.8630, Z -2.1667, A 0.000, B 0.000, C 0.000 }
gfCNCPoint1[26845] = {X -4.6247, Y 10.9722, Z -2.1667, A 0.000, B 0.000, C 0.000 }
gfCNCPoint1[26846] = {X -7.6965, Y 10.9722, Z -2.1667, A 0.000, B 0.000, C 0.000 }
gfCNCPoint1[26847] = {X -7.6965, Y 10.9722, Z 0.8333, A 0.000, B 0.000, C 0.000 }
gfCNCPoint1[26848] = {X -7.6965, Y 10.9722, Z 11.0000, A 0.000, B 0.000, C 0.000 }
gfCNCPoint1[26849] = {X -8.0030, Y 35.5763, Z 11.0000, A 0.000, B 0.000, C 0.000 }
gfCNCPoint1[26850] = {X -8.0030, Y 35.5763, Z 0.8333, A 0.000, B 0.000, C 0.000 }
gfCNCPoint1[26851] = {X -8.0030, Y 35.5763, Z -2.1667, A 0.000, B 0.000, C 0.000 }
gfCNCPoint1[26852] = {X -4.7110, Y 35.5247, Z -2.1667, A 0.000, B 0.000, C 0.000 }
gfCNCPoint1[26853] = {X -3.6965, Y 31.6554, Z -2.1667, A 0.000, B 0.000, C 0.000 }
gfCNCPoint1[26854] = {X -3.5878, Y 31.2638, Z -2.1667, A 0.000, B 0.000, C 0.000 }
gfCNCPoint1[26855] = {X -3.4682, Y 30.8754, Z -2.1667, A 0.000, B 0.000, C 0.000 }
gfCNCPoint1[26856] = {X -3.1436, Y 29.9764, Z -2.1667, A 0.000, B 0.000, C 0.000 }
gfCNCPoint1[26857] = {X -2.7598, Y 29.1009, Z -2.1667, A 0.000, B 0.000, C 0.000 }
gfCNCPoint1[26858] = {X -1.9738, Y 27.7361, Z -2.1667, A 0.000, B 0.000, C 0.000 }
gfCNCPoint1[26859] = {X -0.9934, Y 26.5033, Z -2.1667, A 0.000, B 0.000, C 0.000 }
gfCNCPoint1[26860] = {X 0.1594, Y 25.4302, Z -2.1667, A 0.000, B 0.000, C 0.000 }
gfCNCPoint1[26861] = {X 1.4590, Y 24.5405, Z -2.1667, A 0.000, B 0.000, C 0.000 }
gfCNCPoint1[26862] = {X 1.6922, Y 24.4091, Z -2.1667, A 0.000, B 0.000, C 0.000 }
gfCNCPoint1[26863] = {X 1.9286, Y 24.2838, Z -2.1667, A 0.000, B 0.000, C 0.000 }
gfCNCPoint1[26864] = {X 1.0583, Y 23.9329, Z -2.1667, A 0.000, B 0.000, C 0.000 }
gfCNCPoint1[26865] = {X 0.2888, Y 23.3959, Z -2.1667, A 0.000, B 0.000, C 0.000 }
gfCNCPoint1[26866] = {X -0.3408, Y 22.7001, Z -2.1667, A 0.000, B 0.000, C 0.000 }
gfCNCPoint1[26867] = {X -0.7984, Y 21.8809, Z -2.1667, A 0.000, B 0.000, C 0.000 }
gfCNCPoint1[26868] = {X -3.4715, Y 15.3286, Z -2.1667, A 0.000, B 0.000, C 0.000 }
gfCNCPoint1[26869] = {X -3.6095, Y 14.8822, Z -2.1667, A 0.000, B 0.000, C 0.000 }
gfCNCPoint1[26870] = {X -3.6965, Y 14.4232, Z -2.1667, A 0.000, B 0.000, C 0.000 }
gfCNCPoint1[26871] = {X -4.2196, Y 10.4576, Z -2.1667, A 0.000, B 0.000, C 0.000 }
gfCNCPoint1[26872] = {X -7.6965, Y 10.4576, Z -2.1667, A 0.000, B 0.000, C 0.000 }
gfCNCPoint1[26873] = {X -7.6965, Y 10.4576, Z 0.8333, A 0.000, B 0.000, C 0.000 }
gfCNCPoint1[26874] = {X -7.6965, Y 10.4576, Z 11.0000, A 0.000, B 0.000, C 0.000 }
gfCNCPoint1[26875] = {X -7.9911, Y 36.0089, Z 11.0000, A 0.000, B 0.000, C 0.000 }
gfCNCPoint1[26876] = {X -7.9911, Y 36.0089, Z 0.8333, A 0.000, B 0.000, C 0.000 }
gfCNCPoint1[26877] = {X -7.9911, Y 36.0089, Z -2.1667, A 0.000, B 0.000, C 0.000 }
gfCNCPoint1[26878] = {X -4.6242, Y 35.8758, Z -2.1667, A 0.000, B 0.000, C 0.000 }
gfCNCPoint1[26879] = {X -3.6965, Y 31.9849, Z -2.1667, A 0.000, B 0.000, C 0.000 }
gfCNCPoint1[26880] = {X -3.5550, Y 31.4395, Z -2.1667, A 0.000, B 0.000, C 0.000 }
gfCNCPoint1[26881] = {X -3.3920, Y 30.9001, Z -2.1667, A 0.000, B 0.000, C 0.000 }
gfCNCPoint1[26882] = {X -3.0693, Y 30.0060, Z -2.1667, A 0.000, B 0.000, C 0.000 }
gfCNCPoint1[26883] = {X -2.6877, Y 29.1355, Z -2.1667, A 0.000, B 0.000, C 0.000 }
gfCNCPoint1[26884] = {X -1.9076, Y 27.7810, Z -2.1667, A 0.000, B 0.000, C 0.000 }
gfCNCPoint1[26885] = {X -0.9347, Y 26.5576, Z -2.1667, A 0.000, B 0.000, C 0.000 }
gfCNCPoint1[26886] = {X 0.2094, Y 25.4926, Z -2.1667, A 0.000, B 0.000, C 0.000 }
gfCNCPoint1[26887] = {X 1.4992, Y 24.6097, Z -2.1667, A 0.000, B 0.000, C 0.000 }
gfCNCPoint1[26888] = {X 1.8253, Y 24.4282, Z -2.1667, A 0.000, B 0.000, C 0.000 }
gfCNCPoint1[26889] = {X 2.1577, Y 24.2584, Z -2.1667, A 0.000, B 0.000, C 0.000 }
gfCNCPoint1[26890] = {X 1.2391, Y 23.9362, Z -2.1667, A 0.000, B 0.000, C 0.000 }
gfCNCPoint1[26891] = {X 0.4229, Y 23.4056, Z -2.1667, A 0.000, B 0.000, C 0.000 }
gfCNCPoint1[26892] = {X -0.2443, Y 22.6968, Z -2.1667, A 0.000, B 0.000, C 0.000 }
gfCNCPoint1[26893] = {X -0.7246, Y 21.8500, Z -2.1667, A 0.000, B 0.000, C 0.000 }
gfCNCPoint1[26894] = {X -3.3965, Y 15.3007, Z -2.1667, A 0.000, B 0.000, C 0.000 }
gfCNCPoint1[26895] = {X -3.6235, Y 14.3620, Z -2.1667, A 0.000, B 0.000, C 0.000 }
gfCNCPoint1[26896] = {X -3.6235, Y 13.3962, Z -2.1667, A 0.000, B 0.000, C 0.000 }
gfCNCPoint1[26897] = {X -3.3965, Y 12.4575, Z -2.1667, A 0.000, B 0.000, C 0.000 }
gfCNCPoint1[26898] = {X -2.9669, Y 11.6158, Z -2.1667, A 0.000, B 0.000, C 0.000 }
gfCNCPoint1[26899] = {X -2.3551, Y 10.8955, Z -2.1667, A 0.000, B 0.000, C 0.000 }
gfCNCPoint1[26900] = {X -1.5940, Y 10.3353, Z -2.1667, A 0.000, B 0.000, C 0.000 }
gfCNCPoint1[26901] = {X -0.9968, Y 9.9946, Z -2.1667, A 0.000, B 0.000, C 0.000 }
gfCNCPoint1[26902] = {X -0.1674, Y 9.6366, Z -2.1667, A 0.000, B 0.000, C 0.000 }
gfCNCPoint1[26903] = {X 0.7205, Y 9.4698, Z -2.1667, A 0.000, B 0.000, C 0.000 }
gfCNCPoint1[26904] = {X 1.6233, Y 9.5026, Z -2.1667, A 0.000, B 0.000, C 0.000 }
gfCNCPoint1[26905] = {X 2.4967, Y 9.7332, Z -2.1667, A 0.000, B 0.000, C 0.000 }
gfCNCPoint1[26906] = {X 2.5619, Y 9.7591, Z -2.1667, A 0.000, B 0.000, C 0.000 }
gfCNCPoint1[26907] = {X 2.6267, Y 9.7861, Z -2.1667, A 0.000, B 0.000, C 0.000 }
gfCNCPoint1[26908] = {X 3.4422, Y 9.4007, Z -2.1667, A 0.000, B 0.000, C 0.000 }
gfCNCPoint1[26909] = {X 4.2810, Y 9.0693, Z -2.1667, A 0.000, B 0.000, C 0.000 }
gfCNCPoint1[26910] = {X 6.1732, Y 8.4069, Z -2.1667, A 0.000, B 0.000, C 0.000 }
gfCNCPoint1[26911] = {X 8.1154, Y 7.9101, Z -2.1667, A 0.000, B 0.000, C 0.000 }
gfCNCPoint1[26912] = {X 10.0932, Y 7.5827, Z -2.1667, A 0.000, B 0.000, C 0.000 }
gfCNCPoint1[26913] = {X 12.0919, Y 7.4270, Z -2.1667, A 0.000, B 0.000, C 0.000 }
gfCNCPoint1[26914] = {X 14.0966, Y 7.4442, Z -2.1667, A 0.000, B 0.000, C 0.000 }
gfCNCPoint1[26915] = {X 16.0923, Y 7.6343, Z -2.1667, A 0.000, B 0.000, C 0.000 }
gfCNCPoint1[26916] = {X 17.8907, Y 7.9633, Z -2.1667, A 0.000, B 0.000, C 0.000 }
gfCNCPoint1[26917] = {X 19.6441, Y 8.4812, Z -2.1667, A 0.000, B 0.000, C 0.000 }
gfCNCPoint1[26918] = {X 21.3327, Y 9.1820, Z -2.1667, A 0.000, B 0.000, C 0.000 }
gfCNCPoint1[26919] = {X 22.9375, Y 10.0579, Z -2.1667, A 0.000, B 0.000, C 0.000 }
gfCNCPoint1[26920] = {X 24.4404, Y 11.0991, Z -2.1667, A 0.000, B 0.000, C 0.000 }
gfCNCPoint1[26921] = {X 25.5047, Y 12.0305, Z -2.1667, A 0.000, B 0.000, C 0.000 }
gfCNCPoint1[26922] = {X 26.4595, Y 13.0738, Z -2.1667, A 0.000, B 0.000, C 0.000 }
gfCNCPoint1[26923] = {X 27.2932, Y 14.2163, Z -2.1667, A 0.000, B 0.000, C 0.000 }
gfCNCPoint1[26924] = {X 27.9955, Y 15.4439, Z -2.1667, A 0.000, B 0.000, C 0.000 }
gfCNCPoint1[26925] = {X 28.5578, Y 16.7417, Z -2.1667, A 0.000, B 0.000, C 0.000 }
gfCNCPoint1[26926] = {X 29.0253, Y 18.3710, Z -2.1667, A 0.000, B 0.000, C 0.000 }
gfCNCPoint1[26927] = {X 29.3026, Y 20.0433, Z -2.1667, A 0.000, B 0.000, C 0.000 }
gfCNCPoint1[26928] = {X 29.3860, Y 21.7364, Z -2.1667, A 0.000, B 0.000, C 0.000 }
gfCNCPoint1[26929] = {X 29.2744, Y 23.4278, Z -2.1667, A 0.000, B 0.000, C 0.000 }
gfCNCPoint1[26930] = {X 28.9692, Y 25.0952, Z -2.1667, A 0.000, B 0.000, C 0.000 }
gfCNCPoint1[26931] = {X 28.5018, Y 26.6021, Z -2.1667, A 0.000, B 0.000, C 0.000 }
gfCNCPoint1[26932] = {X 27.8315, Y 28.0303, Z -2.1667, A 0.000, B 0.000, C 0.000 }
gfCNCPoint1[26933] = {X 26.9713, Y 29.3528, Z -2.1667, A 0.000, B 0.000, C 0.000 }
gfCNCPoint1[26934] = {X 25.9374, Y 30.5445, Z -2.1667, A 0.000, B 0.000, C 0.000 }
gfCNCPoint1[26935] = {X 24.7494, Y 31.5828, Z -2.1667, A 0.000, B 0.000, C 0.000 }
gfCNCPoint1[26936] = {X 25.0465, Y 31.6498, Z -2.1667, A 0.000, B 0.000, C 0.000 }
gfCNCPoint1[26937] = {X 25.3377, Y 31.7388, Z -2.1667, A 0.000, B 0.000, C 0.000 }
gfCNCPoint1[26938] = {X 26.0570, Y 32.0697, Z -2.1667, A 0.000, B 0.000, C 0.000 }
gfCNCPoint1[26939] = {X 26.6989, Y 32.5333, Z -2.1667, A 0.000, B 0.000, C 0.000 }
gfCNCPoint1[26940] = {X 27.2392, Y 33.1122, Z -2.1667, A 0.000, B 0.000, C 0.000 }
gfCNCPoint1[26941] = {X 27.6575, Y 33.7845, Z -2.1667, A 0.000, B 0.000, C 0.000 }
gfCNCPoint1[26942] = {X 30.6940, Y 40.0576, Z -2.1667, A 0.000, B 0.000, C 0.000 }
gfCNCPoint1[26943] = {X 30.9967, Y 40.9162, Z -2.1667, A 0.000, B 0.000, C 0.000 }
gfCNCPoint1[26944] = {X 31.1015, Y 41.8206, Z -2.1667, A 0.000, B 0.000, C 0.000 }
gfCNCPoint1[26945] = {X 31.0032, Y 42.7257, Z -2.1667, A 0.000, B 0.000, C 0.000 }
gfCNCPoint1[26946] = {X 30.7066, Y 43.5864, Z -2.1667, A 0.000, B 0.000, C 0.000 }
gfCNCPoint1[26947] = {X 30.2265, Y 44.3600, Z -2.1667, A 0.000, B 0.000, C 0.000 }
gfCNCPoint1[26948] = {X 29.5868, Y 45.0078, Z -2.1667, A 0.000, B 0.000, C 0.000 }
gfCNCPoint1[26949] = {X 29.0507, Y 45.4413, Z -2.1667, A 0.000, B 0.000, C 0.000 }
gfCNCPoint1[26950] = {X 28.3667, Y 45.8883, Z -2.1667, A 0.000, B 0.000, C 0.000 }
gfCNCPoint1[26951] = {X 27.6075, Y 46.1906, Z -2.1667, A 0.000, B 0.000, C 0.000 }
gfCNCPoint1[26952] = {X 26.8035, Y 46.3363, Z -2.1667, A 0.000, B 0.000, C 0.000 }
gfCNCPoint1[26953] = {X 25.9865, Y 46.3196, Z -2.1667, A 0.000, B 0.000, C 0.000 }
gfCNCPoint1[26954] = {X 25.1891, Y 46.1412, Z -2.1667, A 0.000, B 0.000, C 0.000 }
gfCNCPoint1[26955] = {X 23.1601, Y 47.2127, Z -2.1667, A 0.000, B 0.000, C 0.000 }
gfCNCPoint1[26956] = {X 21.0508, Y 48.1163, Z -2.1667, A 0.000, B 0.000, C 0.000 }
gfCNCPoint1[26957] = {X 18.8752, Y 48.8458, Z -2.1667, A 0.000, B 0.000, C 0.000 }
gfCNCPoint1[26958] = {X 16.7975, Y 49.3592, Z -2.1667, A 0.000, B 0.000, C 0.000 }
gfCNCPoint1[26959] = {X 14.6804, Y 49.6718, Z -2.1667, A 0.000, B 0.000, C 0.000 }
gfCNCPoint1[26960] = {X 12.5430, Y 49.7809, Z -2.1667, A 0.000, B 0.000, C 0.000 }
gfCNCPoint1[26961] = {X 10.4050, Y 49.6855, Z -2.1667, A 0.000, B 0.000, C 0.000 }
gfCNCPoint1[26962] = {X 8.2859, Y 49.3864, Z -2.1667, A 0.000, B 0.000, C 0.000 }
gfCNCPoint1[26963] = {X 6.4786, Y 48.9504, Z -2.1667, A 0.000, B 0.000, C 0.000 }
gfCNCPoint1[26964] = {X 4.7302, Y 48.3183, Z -2.1667, A 0.000, B 0.000, C 0.000 }
gfCNCPoint1[26965] = {X 3.0620, Y 47.4977, Z -2.1667, A 0.000, B 0.000, C 0.000 }
gfCNCPoint1[26966] = {X 1.4942, Y 46.4986, Z -2.1667, A 0.000, B 0.000, C 0.000 }
gfCNCPoint1[26967] = {X 0.1924, Y 45.4508, Z -2.1667, A 0.000, B 0.000, C 0.000 }
gfCNCPoint1[26968] = {X -0.9648, Y 44.2452, Z -2.1667, A 0.000, B 0.000, C 0.000 }
gfCNCPoint1[26969] = {X -1.9583, Y 42.9016, Z -2.1667, A 0.000, B 0.000, C 0.000 }
gfCNCPoint1[26970] = {X -2.7720, Y 41.4420, Z -2.1667, A 0.000, B 0.000, C 0.000 }
gfCNCPoint1[26971] = {X -3.3924, Y 39.8903, Z -2.1667, A 0.000, B 0.000, C 0.000 }
gfCNCPoint1[26972] = {X -3.5562, Y 39.3505, Z -2.1667, A 0.000, B 0.000, C 0.000 }
gfCNCPoint1[26973] = {X -3.6965, Y 38.8042, Z -2.1667, A 0.000, B 0.000, C 0.000 }
gfCNCPoint1[26974] = {X -4.6075, Y 34.9093, Z -2.1667, A 0.000, B 0.000, C 0.000 }
gfCNCPoint1[26975] = {X -7.9991, Y 34.8216, Z -2.1667, A 0.000, B 0.000, C 0.000 }
gfCNCPoint1[26976] = {X -7.9991, Y 34.8216, Z 0.8333, A 0.000, B 0.000, C 0.000 }
gfCNCPoint1[26977] = {X -7.9991, Y 34.8216, Z 11.0000, A 0.000, B 0.000, C 0.000 }
gfCNCPoint1[26978] = {X -7.9657, Y 36.4889, Z 11.0000, A 0.000, B 0.000, C 0.000 }
gfCNCPoint1[26979] = {X -7.9657, Y 36.4889, Z 0.8333, A 0.000, B 0.000, C 0.000 }
gfCNCPoint1[26980] = {X -7.9657, Y 36.4889, Z -2.1667, A 0.000, B 0.000, C 0.000 }
gfCNCPoint1[26981] = {X -4.5267, Y 36.2618, Z -2.1667, A 0.000, B 0.000, C 0.000 }
gfCNCPoint1[26982] = {X -3.6965, Y 32.3489, Z -2.1667, A 0.000, B 0.000, C 0.000 }
gfCNCPoint1[26983] = {X -3.5247, Y 31.6319, Z -2.1667, A 0.000, B 0.000, C 0.000 }
gfCNCPoint1[26984] = {X -3.3159, Y 30.9247, Z -2.1667, A 0.000, B 0.000, C 0.000 }
gfCNCPoint1[26985] = {X -2.9950, Y 30.0357, Z -2.1667, A 0.000, B 0.000, C 0.000 }
gfCNCPoint1[26986] = {X -2.6155, Y 29.1700, Z -2.1667, A 0.000, B 0.000, C 0.000 }
gfCNCPoint1[26987] = {X -1.8414, Y 27.8259, Z -2.1667, A 0.000, B 0.000, C 0.000 }
gfCNCPoint1[26988] = {X -0.8759, Y 26.6119, Z -2.1667, A 0.000, B 0.000, C 0.000 }
gfCNCPoint1[26989] = {X 0.2594, Y 25.5551, Z -2.1667, A 0.000, B 0.000, C 0.000 }
gfCNCPoint1[26990] = {X 1.5393, Y 24.6789, Z -2.1667, A 0.000, B 0.000, C 0.000 }
gfCNCPoint1[26991] = {X 1.9712, Y 24.4419, Z -2.1667, A 0.000, B 0.000, C 0.000 }
gfCNCPoint1[26992] = {X 2.4138, Y 24.2256, Z -2.1667, A 0.000, B 0.000, C 0.000 }
gfCNCPoint1[26993] = {X 1.6217, Y 24.0152, Z -2.1667, A 0.000, B 0.000, C 0.000 }
gfCNCPoint1[26994] = {X 0.8891, Y 23.6478, Z -2.1667, A 0.000, B 0.000, C 0.000 }
gfCNCPoint1[26995] = {X 0.2468, Y 23.1389, Z -2.1667, A 0.000, B 0.000, C 0.000 }
gfCNCPoint1[26996] = {X -0.2784, Y 22.5096, Z -2.1667, A 0.000, B 0.000, C 0.000 }
gfCNCPoint1[26997] = {X -0.6642, Y 21.7866, Z -2.1667, A 0.000, B 0.000, C 0.000 }
gfCNCPoint1[26998] = {X -3.2754, Y 15.3911, Z -2.1667, A 0.000, B 0.000, C 0.000 }
gfCNCPoint1[26999] = {X -3.2990, Y 15.3322, Z -2.1667, A 0.000, B 0.000, C 0.000 }
gfCNCPoint1[27000] = {X -3.3216, Y 15.2729, Z -2.1667, A 0.000, B 0.000, C 0.000 }
gfCNCPoint1[27001] = {X -3.5441, Y 14.3525, Z -2.1667, A 0.000, B 0.000, C 0.000 }
gfCNCPoint1[27002] = {X -3.5441, Y 13.4057, Z -2.1667, A 0.000, B 0.000, C 0.000 }
gfCNCPoint1[27003] = {X -3.3216, Y 12.4854, Z -2.1667, A 0.000, B 0.000, C 0.000 }
gfCNCPoint1[27004] = {X -2.9003, Y 11.6602, Z -2.1667, A 0.000, B 0.000, C 0.000 }
gfCNCPoint1[27005] = {X -2.3005, Y 10.9540, Z -2.1667, A 0.000, B 0.000, C 0.000 }
gfCNCPoint1[27006] = {X -1.5544, Y 10.4048, Z -2.1667, A 0.000, B 0.000, C 0.000 }
gfCNCPoint1[27007] = {X -0.9063, Y 10.0355, Z -2.1667, A 0.000, B 0.000, C 0.000 }
gfCNCPoint1[27008] = {X -0.1021, Y 9.7005, Z -2.1667, A 0.000, B 0.000, C 0.000 }
gfCNCPoint1[27009] = {X 0.7555, Y 9.5475, Z -2.1667, A 0.000, B 0.000, C 0.000 }
gfCNCPoint1[27010] = {X 1.6260, Y 9.5839, Z -2.1667, A 0.000, B 0.000, C 0.000 }
gfCNCPoint1[27011] = {X 2.4679, Y 9.8078, Z -2.1667, A 0.000, B 0.000, C 0.000 }
gfCNCPoint1[27012] = {X 2.5491, Y 9.8403, Z -2.1667, A 0.000, B 0.000, C 0.000 }
gfCNCPoint1[27013] = {X 2.6297, Y 9.8745, Z -2.1667, A 0.000, B 0.000, C 0.000 }
gfCNCPoint1[27014] = {X 3.4606, Y 9.4798, Z -2.1667, A 0.000, B 0.000, C 0.000 }
gfCNCPoint1[27015] = {X 4.3160, Y 9.1415, Z -2.1667, A 0.000, B 0.000, C 0.000 }
gfCNCPoint1[27016] = {X 6.2009, Y 8.4821, Z -2.1667, A 0.000, B 0.000, C 0.000 }
gfCNCPoint1[27017] = {X 8.1357, Y 7.9876, Z -2.1667, A 0.000, B 0.000, C 0.000 }
gfCNCPoint1[27018] = {X 10.1058, Y 7.6617, Z -2.1667, A 0.000, B 0.000, C 0.000 }
gfCNCPoint1[27019] = {X 12.0968, Y 7.5069, Z -2.1667, A 0.000, B 0.000, C 0.000 }
gfCNCPoint1[27020] = {X 14.0936, Y 7.5242, Z -2.1667, A 0.000, B 0.000, C 0.000 }
gfCNCPoint1[27021] = {X 16.0816, Y 7.7136, Z -2.1667, A 0.000, B 0.000, C 0.000 }
gfCNCPoint1[27022] = {X 16.4808, Y 7.7686, Z -2.1667, A 0.000, B 0.000, C 0.000 }
gfCNCPoint1[27023] = {X 18.1848, Y 8.1179, Z -2.1667, A 0.000, B 0.000, C 0.000 }
gfCNCPoint1[27024] = {X 19.8447, Y 8.6382, Z -2.1667, A 0.000, B 0.000, C 0.000 }
gfCNCPoint1[27025] = {X 21.4432, Y 9.3239, Z -2.1667, A 0.000, B 0.000, C 0.000 }
gfCNCPoint1[27026] = {X 22.9640, Y 10.1682, Z -2.1667, A 0.000, B 0.000, C 0.000 }
gfCNCPoint1[27027] = {X 24.3914, Y 11.1623, Z -2.1667, A 0.000, B 0.000, C 0.000 }
gfCNCPoint1[27028] = {X 25.4488, Y 12.0878, Z -2.1667, A 0.000, B 0.000, C 0.000 }
gfCNCPoint1[27029] = {X 26.3975, Y 13.1245, Z -2.1667, A 0.000, B 0.000, C 0.000 }
gfCNCPoint1[27030] = {X 27.2259, Y 14.2596, Z -2.1667, A 0.000, B 0.000, C 0.000 }
gfCNCPoint1[27031] = {X 27.9237, Y 15.4794, Z -2.1667, A 0.000, B 0.000, C 0.000 }
gfCNCPoint1[27032] = {X 28.4825, Y 16.7687, Z -2.1667, A 0.000, B 0.000, C 0.000 }
gfCNCPoint1[27033] = {X 28.9474, Y 18.3895, Z -2.1667, A 0.000, B 0.000, C 0.000 }
gfCNCPoint1[27034] = {X 29.2231, Y 20.0528, Z -2.1667, A 0.000, B 0.000, C 0.000 }
gfCNCPoint1[27035] = {X 29.3060, Y 21.7369, Z -2.1667, A 0.000, B 0.000, C 0.000 }
gfCNCPoint1[27036] = {X 29.1948, Y 23.4193, Z -2.1667, A 0.000, B 0.000, C 0.000 }
gfCNCPoint1[27037] = {X 28.8911, Y 25.0778, Z -2.1667, A 0.000, B 0.000, C 0.000 }
gfCNCPoint1[27038] = {X 28.4132, Y 26.6089, Z -2.1667, A 0.000, B 0.000, C 0.000 }
gfCNCPoint1[27039] = {X 27.7246, Y 28.0575, Z -2.1667, A 0.000, B 0.000, C 0.000 }
gfCNCPoint1[27040] = {X 26.8388, Y 29.3948, Z -2.1667, A 0.000, B 0.000, C 0.000 }
gfCNCPoint1[27041] = {X 25.7737, Y 30.5940, Z -2.1667, A 0.000, B 0.000, C 0.000 }
gfCNCPoint1[27042] = {X 24.5504, Y 31.6314, Z -2.1667, A 0.000, B 0.000, C 0.000 }
gfCNCPoint1[27043] = {X 24.9354, Y 31.7042, Z -2.1667, A 0.000, B 0.000, C 0.000 }
gfCNCPoint1[27044] = {X 25.3114, Y 31.8144, Z -2.1667, A 0.000, B 0.000, C 0.000 }
gfCNCPoint1[27045] = {X 26.0241, Y 32.1431, Z -2.1667, A 0.000, B 0.000, C 0.000 }
gfCNCPoint1[27046] = {X 26.6589, Y 32.6047, Z -2.1667, A 0.000, B 0.000, C 0.000 }
gfCNCPoint1[27047] = {X 27.1913, Y 33.1813, Z -2.1667, A 0.000, B 0.000, C 0.000 }
gfCNCPoint1[27048] = {X 27.6008, Y 33.8508, Z -2.1667, A 0.000, B 0.000, C 0.000 }
gfCNCPoint1[27049] = {X 30.6220, Y 40.0925, Z -2.1667, A 0.000, B 0.000, C 0.000 }
gfCNCPoint1[27050] = {X 30.9188, Y 40.9342, Z -2.1667, A 0.000, B 0.000, C 0.000 }
gfCNCPoint1[27051] = {X 31.0215, Y 41.8209, Z -2.1667, A 0.000, B 0.000, C 0.000 }
gfCNCPoint1[27052] = {X 30.9251, Y 42.7082, Z -2.1667, A 0.000, B 0.000, C 0.000 }
gfCNCPoint1[27053] = {X 30.6343, Y 43.5521, Z -2.1667, A 0.000, B 0.000, C 0.000 }
gfCNCPoint1[27054] = {X 30.1637, Y 44.3105, Z -2.1667, A 0.000, B 0.000, C 0.000 }
gfCNCPoint1[27055] = {X 29.5365, Y 44.9456, Z -2.1667, A 0.000, B 0.000, C 0.000 }
gfCNCPoint1[27056] = {X 29.0005, Y 45.3790, Z -2.1667, A 0.000, B 0.000, C 0.000 }
gfCNCPoint1[27057] = {X 28.3234, Y 45.8206, Z -2.1667, A 0.000, B 0.000, C 0.000 }
gfCNCPoint1[27058] = {X 27.5717, Y 46.1177, Z -2.1667, A 0.000, B 0.000, C 0.000 }
gfCNCPoint1[27059] = {X 26.7756, Y 46.2582, Z -2.1667, A 0.000, B 0.000, C 0.000 }
gfCNCPoint1[27060] = {X 25.9676, Y 46.2367, Z -2.1667, A 0.000, B 0.000, C 0.000 }
gfCNCPoint1[27061] = {X 25.1802, Y 46.0538, Z -2.1667, A 0.000, B 0.000, C 0.000 }
gfCNCPoint1[27062] = {X 25.1044, Y 46.0978, Z -2.1667, A 0.000, B 0.000, C 0.000 }
gfCNCPoint1[27063] = {X 25.0283, Y 46.1417, Z -2.1667, A 0.000, B 0.000, C 0.000 }
gfCNCPoint1[27064] = {X 23.0413, Y 47.1806, Z -2.1667, A 0.000, B 0.000, C 0.000 }
gfCNCPoint1[27065] = {X 20.9780, Y 48.0583, Z -2.1667, A 0.000, B 0.000, C 0.000 }
gfCNCPoint1[27066] = {X 18.8515, Y 48.7694, Z -2.1667, A 0.000, B 0.000, C 0.000 }
gfCNCPoint1[27067] = {X 16.9517, Y 49.2465, Z -2.1667, A 0.000, B 0.000, C 0.000 }
gfCNCPoint1[27068] = {X 15.0173, Y 49.5552, Z -2.1667, A 0.000, B 0.000, C 0.000 }
gfCNCPoint1[27069] = {X 13.0633, Y 49.6931, Z -2.1667, A 0.000, B 0.000, C 0.000 }
gfCNCPoint1[27070] = {X 11.1047, Y 49.6590, Z -2.1667, A 0.000, B 0.000, C 0.000 }
gfCNCPoint1[27071] = {X 9.1567, Y 49.4532, Z -2.1667, A 0.000, B 0.000, C 0.000 }
gfCNCPoint1[27072] = {X 8.4642, Y 49.3343, Z -2.1667, A 0.000, B 0.000, C 0.000 }
gfCNCPoint1[27073] = {X 8.3003, Y 49.3077, Z -2.1667, A 0.000, B 0.000, C 0.000 }
gfCNCPoint1[27074] = {X 6.5012, Y 48.8736, Z -2.1667, A 0.000, B 0.000, C 0.000 }
gfCNCPoint1[27075] = {X 4.7607, Y 48.2443, Z -2.1667, A 0.000, B 0.000, C 0.000 }
gfCNCPoint1[27076] = {X 3.1001, Y 47.4273, Z -2.1667, A 0.000, B 0.000, C 0.000 }
gfCNCPoint1[27077] = {X 1.5394, Y 46.4325, Z -2.1667, A 0.000, B 0.000, C 0.000 }
gfCNCPoint1[27078] = {X 0.2458, Y 45.3912, Z -2.1667, A 0.000, B 0.000, C 0.000 }
gfCNCPoint1[27079] = {X -0.9040, Y 44.1931, Z -2.1667, A 0.000, B 0.000, C 0.000 }
gfCNCPoint1[27080] = {X -1.8913, Y 42.8579, Z -2.1667, A 0.000, B 0.000, C 0.000 }
gfCNCPoint1[27081] = {X -2.6998, Y 41.4074, Z -2.1667, A 0.000, B 0.000, C 0.000 }
gfCNCPoint1[27082] = {X -3.3163, Y 39.8654, Z -2.1667, A 0.000, B 0.000, C 0.000 }
gfCNCPoint1[27083] = {X -3.5270, Y 39.1534, Z -2.1667, A 0.000, B 0.000, C 0.000 }
gfCNCPoint1[27084] = {X -3.6965, Y 38.4305, Z -2.1667, A 0.000, B 0.000, C 0.000 }
gfCNCPoint1[27085] = {X -4.4979, Y 34.5116, Z -2.1667, A 0.000, B 0.000, C 0.000 }
gfCNCPoint1[27086] = {X -7.9796, Y 34.3265, Z -2.1667, A 0.000, B 0.000, C 0.000 }
gfCNCPoint1[27087] = {X -7.9796, Y 34.3265, Z 0.8333, A 0.000, B 0.000, C 0.000 }
gfCNCPoint1[27088] = {X -7.9796, Y 34.3265, Z 11.0000, A 0.000, B 0.000, C 0.000 }
gfCNCPoint1[27089] = {X 39.8140, Y 26.4139, Z 11.0000, A 0.000, B 0.000, C 0.000 }
gfCNCPoint1[27090] = {X 39.8140, Y 26.4139, Z 0.8333, A 0.000, B 0.000, C 0.000 }
gfCNCPoint1[27091] = {X 39.8140, Y 26.4139, Z -2.1667, A 0.000, B 0.000, C 0.000 }
gfCNCPoint1[27092] = {X 43.6374, Y 27.8378, Z -2.1667, A 0.000, B 0.000, C 0.000 }
gfCNCPoint1[27093] = {X 48.2902, Y 15.3446, Z -2.1667, A 0.000, B 0.000, C 0.000 }
gfCNCPoint1[27094] = {X 47.9079, Y 14.6186, Z -2.1667, A 0.000, B 0.000, C 0.000 }
gfCNCPoint1[27095] = {X 47.6698, Y 13.8334, Z -2.1667, A 0.000, B 0.000, C 0.000 }
gfCNCPoint1[27096] = {X 47.5844, Y 13.0173, Z -2.1667, A 0.000, B 0.000, C 0.000 }
gfCNCPoint1[27097] = {X 47.5842, Y 12.1868, Z -2.1667, A 0.000, B 0.000, C 0.000 }
gfCNCPoint1[27098] = {X 47.6925, Y 11.2255, Z -2.1667, A 0.000, B 0.000, C 0.000 }
gfCNCPoint1[27099] = {X 48.0120, Y 10.3125, Z -2.1667, A 0.000, B 0.000, C 0.000 }
gfCNCPoint1[27100] = {X 48.5267, Y 9.4933, Z -2.1667, A 0.000, B 0.000, C 0.000 }
gfCNCPoint1[27101] = {X 49.2107, Y 8.8093, Z -2.1667, A 0.000, B 0.000, C 0.000 }
gfCNCPoint1[27102] = {X 50.0298, Y 8.2946, Z -2.1667, A 0.000, B 0.000, C 0.000 }
gfCNCPoint1[27103] = {X 50.9429, Y 7.9751, Z -2.1667, A 0.000, B 0.000, C 0.000 }
gfCNCPoint1[27104] = {X 51.9042, Y 7.8668, Z -2.1667, A 0.000, B 0.000, C 0.000 }
gfCNCPoint1[27105] = {X 59.6221, Y 7.8668, Z -2.1667, A 0.000, B 0.000, C 0.000 }
gfCNCPoint1[27106] = {X 60.5834, Y 7.9751, Z -2.1667, A 0.000, B 0.000, C 0.000 }
gfCNCPoint1[27107] = {X 61.4965, Y 8.2946, Z -2.1667, A 0.000, B 0.000, C 0.000 }
gfCNCPoint1[27108] = {X 62.3156, Y 8.8093, Z -2.1667, A 0.000, B 0.000, C 0.000 }
gfCNCPoint1[27109] = {X 62.9996, Y 9.4933, Z -2.1667, A 0.000, B 0.000, C 0.000 }
gfCNCPoint1[27110] = {X 63.5143, Y 10.3124, Z -2.1667, A 0.000, B 0.000, C 0.000 }
gfCNCPoint1[27111] = {X 63.8338, Y 11.2255, Z -2.1667, A 0.000, B 0.000, C 0.000 }
gfCNCPoint1[27112] = {X 63.9421, Y 12.1868, Z -2.1667, A 0.000, B 0.000, C 0.000 }
gfCNCPoint1[27113] = {X 63.9421, Y 12.9781, Z -2.1667, A 0.000, B 0.000, C 0.000 }
gfCNCPoint1[27114] = {X 63.8583, Y 13.8248, Z -2.1667, A 0.000, B 0.000, C 0.000 }
gfCNCPoint1[27115] = {X 63.6102, Y 14.6386, Z -2.1667, A 0.000, B 0.000, C 0.000 }
gfCNCPoint1[27116] = {X 63.2074, Y 15.3880, Z -2.1667, A 0.000, B 0.000, C 0.000 }
gfCNCPoint1[27117] = {X 63.4697, Y 16.0735, Z -2.1667, A 0.000, B 0.000, C 0.000 }
gfCNCPoint1[27118] = {X 66.0342, Y 22.8875, Z -2.1667, A 0.000, B 0.000, C 0.000 }
gfCNCPoint1[27119] = {X 72.2087, Y 39.5004, Z -2.1667, A 0.000, B 0.000, C 0.000 }
gfCNCPoint1[27120] = {X 72.5138, Y 40.2677, Z -2.1667, A 0.000, B 0.000, C 0.000 }
gfCNCPoint1[27121] = {X 73.3585, Y 40.7694, Z -2.1667, A 0.000, B 0.000, C 0.000 }
gfCNCPoint1[27122] = {X 74.0681, Y 41.4491, Z -2.1667, A 0.000, B 0.000, C 0.000 }
gfCNCPoint1[27123] = {X 74.6057, Y 42.2715, Z -2.1667, A 0.000, B 0.000, C 0.000 }
gfCNCPoint1[27124] = {X 74.9436, Y 43.1941, Z -2.1667, A 0.000, B 0.000, C 0.000 }
gfCNCPoint1[27125] = {X 75.0643, Y 44.1692, Z -2.1667, A 0.000, B 0.000, C 0.000 }
gfCNCPoint1[27126] = {X 75.0645, Y 45.0000, Z -2.1667, A 0.000, B 0.000, C 0.000 }
gfCNCPoint1[27127] = {X 74.9561, Y 45.9613, Z -2.1667, A 0.000, B 0.000, C 0.000 }
gfCNCPoint1[27128] = {X 74.6366, Y 46.8744, Z -2.1667, A 0.000, B 0.000, C 0.000 }
gfCNCPoint1[27129] = {X 74.1220, Y 47.6935, Z -2.1667, A 0.000, B 0.000, C 0.000 }
gfCNCPoint1[27130] = {X 73.4379, Y 48.3775, Z -2.1667, A 0.000, B 0.000, C 0.000 }
gfCNCPoint1[27131] = {X 72.6188, Y 48.8922, Z -2.1667, A 0.000, B 0.000, C 0.000 }
gfCNCPoint1[27132] = {X 71.7057, Y 49.2117, Z -2.1667, A 0.000, B 0.000, C 0.000 }
gfCNCPoint1[27133] = {X 70.7445, Y 49.3200, Z -2.1667, A 0.000, B 0.000, C 0.000 }
gfCNCPoint1[27134] = {X 64.1851, Y 49.3200, Z -2.1667, A 0.000, B 0.000, C 0.000 }
gfCNCPoint1[27135] = {X 63.2238, Y 49.2117, Z -2.1667, A 0.000, B 0.000, C 0.000 }
gfCNCPoint1[27136] = {X 62.3108, Y 48.8922, Z -2.1667, A 0.000, B 0.000, C 0.000 }
gfCNCPoint1[27137] = {X 61.4917, Y 48.3775, Z -2.1667, A 0.000, B 0.000, C 0.000 }
gfCNCPoint1[27138] = {X 60.8076, Y 47.6935, Z -2.1667, A 0.000, B 0.000, C 0.000 }
gfCNCPoint1[27139] = {X 60.2930, Y 46.8744, Z -2.1667, A 0.000, B 0.000, C 0.000 }
gfCNCPoint1[27140] = {X 59.9734, Y 45.9613, Z -2.1667, A 0.000, B 0.000, C 0.000 }
gfCNCPoint1[27141] = {X 59.8651, Y 45.0000, Z -2.1667, A 0.000, B 0.000, C 0.000 }
gfCNCPoint1[27142] = {X 59.8651, Y 44.2084, Z -2.1667, A 0.000, B 0.000, C 0.000 }
gfCNCPoint1[27143] = {X 59.9521, Y 43.3499, Z -2.1667, A 0.000, B 0.000, C 0.000 }
gfCNCPoint1[27144] = {X 60.2079, Y 42.5259, Z -2.1667, A 0.000, B 0.000, C 0.000 }
gfCNCPoint1[27145] = {X 60.6224, Y 41.7691, Z -2.1667, A 0.000, B 0.000, C 0.000 }
gfCNCPoint1[27146] = {X 60.0074, Y 40.0892, Z -2.1667, A 0.000, B 0.000, C 0.000 }
gfCNCPoint1[27147] = {X 52.0764, Y 40.0892, Z -2.1667, A 0.000, B 0.000, C 0.000 }
gfCNCPoint1[27148] = {X 51.3339, Y 42.0838, Z -2.1667, A 0.000, B 0.000, C 0.000 }
gfCNCPoint1[27149] = {X 51.3372, Y 42.0891, Z -2.1667, A 0.000, B 0.000, C 0.000 }
gfCNCPoint1[27150] = {X 51.6388, Y 42.7488, Z -2.1667, A 0.000, B 0.000, C 0.000 }
gfCNCPoint1[27151] = {X 51.8257, Y 43.4497, Z -2.1667, A 0.000, B 0.000, C 0.000 }
gfCNCPoint1[27152] = {X 51.8928, Y 44.1720, Z -2.1667, A 0.000, B 0.000, C 0.000 }
gfCNCPoint1[27153] = {X 51.8929, Y 45.0000, Z -2.1667, A 0.000, B 0.000, C 0.000 }
gfCNCPoint1[27154] = {X 51.7846, Y 45.9613, Z -2.1667, A 0.000, B 0.000, C 0.000 }
gfCNCPoint1[27155] = {X 51.4651, Y 46.8744, Z -2.1667, A 0.000, B 0.000, C 0.000 }
gfCNCPoint1[27156] = {X 50.9504, Y 47.6935, Z -2.1667, A 0.000, B 0.000, C 0.000 }
gfCNCPoint1[27157] = {X 50.2664, Y 48.3775, Z -2.1667, A 0.000, B 0.000, C 0.000 }
gfCNCPoint1[27158] = {X 49.4473, Y 48.8922, Z -2.1667, A 0.000, B 0.000, C 0.000 }
gfCNCPoint1[27159] = {X 48.5342, Y 49.2117, Z -2.1667, A 0.000, B 0.000, C 0.000 }
gfCNCPoint1[27160] = {X 47.5729, Y 49.3200, Z -2.1667, A 0.000, B 0.000, C 0.000 }
gfCNCPoint1[27161] = {X 40.6393, Y 49.3200, Z -2.1667, A 0.000, B 0.000, C 0.000 }
gfCNCPoint1[27162] = {X 39.6780, Y 49.2117, Z -2.1667, A 0.000, B 0.000, C 0.000 }
gfCNCPoint1[27163] = {X 38.7649, Y 48.8922, Z -2.1667, A 0.000, B 0.000, C 0.000 }
gfCNCPoint1[27164] = {X 37.9458, Y 48.3775, Z -2.1667, A 0.000, B 0.000, C 0.000 }
gfCNCPoint1[27165] = {X 37.2618, Y 47.6935, Z -2.1667, A 0.000, B 0.000, C 0.000 }
gfCNCPoint1[27166] = {X 36.7471, Y 46.8744, Z -2.1667, A 0.000, B 0.000, C 0.000 }
gfCNCPoint1[27167] = {X 36.4276, Y 45.9613, Z -2.1667, A 0.000, B 0.000, C 0.000 }
gfCNCPoint1[27168] = {X 36.3193, Y 45.0000, Z -2.1667, A 0.000, B 0.000, C 0.000 }
gfCNCPoint1[27169] = {X 36.3193, Y 44.2086, Z -2.1667, A 0.000, B 0.000, C 0.000 }
gfCNCPoint1[27170] = {X 36.4325, Y 43.2261, Z -2.1667, A 0.000, B 0.000, C 0.000 }
gfCNCPoint1[27171] = {X 36.7663, Y 42.2951, Z -2.1667, A 0.000, B 0.000, C 0.000 }
gfCNCPoint1[27172] = {X 37.3031, Y 41.4644, Z -2.1667, A 0.000, B 0.000, C 0.000 }
gfCNCPoint1[27173] = {X 38.0147, Y 40.7775, Z -2.1667, A 0.000, B 0.000, C 0.000 }
gfCNCPoint1[27174] = {X 38.8639, Y 40.2705, Z -2.1667, A 0.000, B 0.000, C 0.000 }
gfCNCPoint1[27175] = {X 38.9647, Y 40.1700, Z -2.1667, A 0.000, B 0.000, C 0.000 }
gfCNCPoint1[27176] = {X 39.5385, Y 38.8090, Z -2.1667, A 0.000, B 0.000, C 0.000 }
gfCNCPoint1[27177] = {X 40.0654, Y 37.4292, Z -2.1667, A 0.000, B 0.000, C 0.000 }
gfCNCPoint1[27178] = {X 43.6374, Y 27.8378, Z -2.1667, A 0.000, B 0.000, C 0.000 }
gfCNCPoint1[27179] = {X 39.8890, Y 26.4418, Z -2.1667, A 0.000, B 0.000, C 0.000 }
gfCNCPoint1[27180] = {X 43.7124, Y 27.8657, Z -2.1667, A 0.000, B 0.000, C 0.000 }
gfCNCPoint1[27181] = {X 48.3793, Y 15.3344, Z -2.1667, A 0.000, B 0.000, C 0.000 }
gfCNCPoint1[27182] = {X 47.9922, Y 14.6130, Z -2.1667, A 0.000, B 0.000, C 0.000 }
gfCNCPoint1[27183] = {X 47.7508, Y 13.8307, Z -2.1667, A 0.000, B 0.000, C 0.000 }
gfCNCPoint1[27184] = {X 47.6644, Y 13.0166, Z -2.1667, A 0.000, B 0.000, C 0.000 }
gfCNCPoint1[27185] = {X 47.6642, Y 12.1868, Z -2.1667, A 0.000, B 0.000, C 0.000 }
gfCNCPoint1[27186] = {X 47.7705, Y 11.2433, Z -2.1667, A 0.000, B 0.000, C 0.000 }
gfCNCPoint1[27187] = {X 48.0841, Y 10.3472, Z -2.1667, A 0.000, B 0.000, C 0.000 }
gfCNCPoint1[27188] = {X 48.5893, Y 9.5432, Z -2.1667, A 0.000, B 0.000, C 0.000 }
gfCNCPoint1[27189] = {X 49.2606, Y 8.8719, Z -2.1667, A 0.000, B 0.000, C 0.000 }
gfCNCPoint1[27190] = {X 50.0646, Y 8.3667, Z -2.1667, A 0.000, B 0.000, C 0.000 }
gfCNCPoint1[27191] = {X 50.9607, Y 8.0531, Z -2.1667, A 0.000, B 0.000, C 0.000 }
gfCNCPoint1[27192] = {X 51.9042, Y 7.9468, Z -2.1667, A 0.000, B 0.000, C 0.000 }
gfCNCPoint1[27193] = {X 59.6221, Y 7.9468, Z -2.1667, A 0.000, B 0.000, C 0.000 }
gfCNCPoint1[27194] = {X 60.5656, Y 8.0531, Z -2.1667, A 0.000, B 0.000, C 0.000 }
gfCNCPoint1[27195] = {X 61.4618, Y 8.3667, Z -2.1667, A 0.000, B 0.000, C 0.000 }
gfCNCPoint1[27196] = {X 62.2657, Y 8.8718, Z -2.1667, A 0.000, B 0.000, C 0.000 }
gfCNCPoint1[27197] = {X 62.9371, Y 9.5432, Z -2.1667, A 0.000, B 0.000, C 0.000 }
gfCNCPoint1[27198] = {X 63.4422, Y 10.3471, Z -2.1667, A 0.000, B 0.000, C 0.000 }
gfCNCPoint1[27199] = {X 63.7558, Y 11.2433, Z -2.1667, A 0.000, B 0.000, C 0.000 }
gfCNCPoint1[27200] = {X 63.8621, Y 12.1868, Z -2.1667, A 0.000, B 0.000, C 0.000 }
gfCNCPoint1[27201] = {X 63.8621, Y 12.9781, Z -2.1667, A 0.000, B 0.000, C 0.000 }
gfCNCPoint1[27202] = {X 63.7772, Y 13.8226, Z -2.1667, A 0.000, B 0.000, C 0.000 }
gfCNCPoint1[27203] = {X 63.5257, Y 14.6333, Z -2.1667, A 0.000, B 0.000, C 0.000 }
gfCNCPoint1[27204] = {X 63.1178, Y 15.3776, Z -2.1667, A 0.000, B 0.000, C 0.000 }
gfCNCPoint1[27205] = {X 63.3949, Y 16.1019, Z -2.1667, A 0.000, B 0.000, C 0.000 }
gfCNCPoint1[27206] = {X 65.9592, Y 22.9155, Z -2.1667, A 0.000, B 0.000, C 0.000 }
gfCNCPoint1[27207] = {X 72.1340, Y 39.5291, Z -2.1667, A 0.000, B 0.000, C 0.000 }
gfCNCPoint1[27208] = {X 72.4515, Y 40.3276, Z -2.1667, A 0.000, B 0.000, C 0.000 }
gfCNCPoint1[27209] = {X 73.2895, Y 40.8176, Z -2.1667, A 0.000, B 0.000, C 0.000 }
gfCNCPoint1[27210] = {X 73.9941, Y 41.4853, Z -2.1667, A 0.000, B 0.000, C 0.000 }
gfCNCPoint1[27211] = {X 74.5284, Y 42.2958, Z -2.1667, A 0.000, B 0.000, C 0.000 }
gfCNCPoint1[27212] = {X 74.8643, Y 43.2066, Z -2.1667, A 0.000, B 0.000, C 0.000 }
gfCNCPoint1[27213] = {X 74.9843, Y 44.1699, Z -2.1667, A 0.000, B 0.000, C 0.000 }
gfCNCPoint1[27214] = {X 74.9845, Y 45.0000, Z -2.1667, A 0.000, B 0.000, C 0.000 }
gfCNCPoint1[27215] = {X 74.8782, Y 45.9435, Z -2.1667, A 0.000, B 0.000, C 0.000 }
gfCNCPoint1[27216] = {X 74.5646, Y 46.8397, Z -2.1667, A 0.000, B 0.000, C 0.000 }
gfCNCPoint1[27217] = {X 74.0594, Y 47.6436, Z -2.1667, A 0.000, B 0.000, C 0.000 }
gfCNCPoint1[27218] = {X 73.3881, Y 48.3150, Z -2.1667, A 0.000, B 0.000, C 0.000 }
gfCNCPoint1[27219] = {X 72.5841, Y 48.8201, Z -2.1667, A 0.000, B 0.000, C 0.000 }
gfCNCPoint1[27220] = {X 71.6879, Y 49.1337, Z -2.1667, A 0.000, B 0.000, C 0.000 }
gfCNCPoint1[27221] = {X 70.7445, Y 49.2400, Z -2.1667, A 0.000, B 0.000, C 0.000 }
gfCNCPoint1[27222] = {X 64.1851, Y 49.2400, Z -2.1667, A 0.000, B 0.000, C 0.000 }
gfCNCPoint1[27223] = {X 63.2416, Y 49.1337, Z -2.1667, A 0.000, B 0.000, C 0.000 }
gfCNCPoint1[27224] = {X 62.3455, Y 48.8201, Z -2.1667, A 0.000, B 0.000, C 0.000 }
gfCNCPoint1[27225] = {X 61.5415, Y 48.3150, Z -2.1667, A 0.000, B 0.000, C 0.000 }
gfCNCPoint1[27226] = {X 60.8702, Y 47.6436, Z -2.1667, A 0.000, B 0.000, C 0.000 }
gfCNCPoint1[27227] = {X 60.3650, Y 46.8397, Z -2.1667, A 0.000, B 0.000, C 0.000 }
gfCNCPoint1[27228] = {X 60.0514, Y 45.9435, Z -2.1667, A 0.000, B 0.000, C 0.000 }
gfCNCPoint1[27229] = {X 59.9451, Y 45.0000, Z -2.1667, A 0.000, B 0.000, C 0.000 }
gfCNCPoint1[27230] = {X 59.9451, Y 44.2085, Z -2.1667, A 0.000, B 0.000, C 0.000 }
gfCNCPoint1[27231] = {X 60.0332, Y 43.3525, Z -2.1667, A 0.000, B 0.000, C 0.000 }
gfCNCPoint1[27232] = {X 60.2923, Y 42.5319, Z -2.1667, A 0.000, B 0.000, C 0.000 }
gfCNCPoint1[27233] = {X 60.7118, Y 41.7805, Z -2.1667, A 0.000, B 0.000, C 0.000 }
gfCNCPoint1[27234] = {X 60.0633, Y 40.0092, Z -2.1667, A 0.000, B 0.000, C 0.000 }
gfCNCPoint1[27235] = {X 52.0209, Y 40.0092, Z -2.1667, A 0.000, B 0.000, C 0.000 }
gfCNCPoint1[27236] = {X 51.2454, Y 42.0922, Z -2.1667, A 0.000, B 0.000, C 0.000 }
gfCNCPoint1[27237] = {X 51.2681, Y 42.1295, Z -2.1667, A 0.000, B 0.000, C 0.000 }
gfCNCPoint1[27238] = {X 51.5638, Y 42.7767, Z -2.1667, A 0.000, B 0.000, C 0.000 }
gfCNCPoint1[27239] = {X 51.7470, Y 43.4642, Z -2.1667, A 0.000, B 0.000, C 0.000 }
gfCNCPoint1[27240] = {X 51.8128, Y 44.1726, Z -2.1667, A 0.000, B 0.000, C 0.000 }
gfCNCPoint1[27241] = {X 51.8129, Y 45.0000, Z -2.1667, A 0.000, B 0.000, C 0.000 }
gfCNCPoint1[27242] = {X 51.7066, Y 45.9435, Z -2.1667, A 0.000, B 0.000, C 0.000 }
gfCNCPoint1[27243] = {X 51.3930, Y 46.8397, Z -2.1667, A 0.000, B 0.000, C 0.000 }
gfCNCPoint1[27244] = {X 50.8879, Y 47.6436, Z -2.1667, A 0.000, B 0.000, C 0.000 }
gfCNCPoint1[27245] = {X 50.2165, Y 48.3150, Z -2.1667, A 0.000, B 0.000, C 0.000 }
gfCNCPoint1[27246] = {X 49.4126, Y 48.8201, Z -2.1667, A 0.000, B 0.000, C 0.000 }
gfCNCPoint1[27247] = {X 48.5164, Y 49.1337, Z -2.1667, A 0.000, B 0.000, C 0.000 }
gfCNCPoint1[27248] = {X 47.5729, Y 49.2400, Z -2.1667, A 0.000, B 0.000, C 0.000 }
gfCNCPoint1[27249] = {X 40.6393, Y 49.2400, Z -2.1667, A 0.000, B 0.000, C 0.000 }
gfCNCPoint1[27250] = {X 39.6958, Y 49.1337, Z -2.1667, A 0.000, B 0.000, C 0.000 }
gfCNCPoint1[27251] = {X 38.7996, Y 48.8201, Z -2.1667, A 0.000, B 0.000, C 0.000 }
gfCNCPoint1[27252] = {X 37.9957, Y 48.3150, Z -2.1667, A 0.000, B 0.000, C 0.000 }
gfCNCPoint1[27253] = {X 37.3243, Y 47.6436, Z -2.1667, A 0.000, B 0.000, C 0.000 }
gfCNCPoint1[27254] = {X 36.8192, Y 46.8397, Z -2.1667, A 0.000, B 0.000, C 0.000 }
gfCNCPoint1[27255] = {X 36.5056, Y 45.9435, Z -2.1667, A 0.000, B 0.000, C 0.000 }
gfCNCPoint1[27256] = {X 36.3993, Y 45.0000, Z -2.1667, A 0.000, B 0.000, C 0.000 }
gfCNCPoint1[27257] = {X 36.3993, Y 44.2086, Z -2.1667, A 0.000, B 0.000, C 0.000 }
gfCNCPoint1[27258] = {X 36.5111, Y 43.2415, Z -2.1667, A 0.000, B 0.000, C 0.000 }
gfCNCPoint1[27259] = {X 36.8406, Y 42.3253, Z -2.1667, A 0.000, B 0.000, C 0.000 }
gfCNCPoint1[27260] = {X 37.3704, Y 41.5085, Z -2.1667, A 0.000, B 0.000, C 0.000 }
gfCNCPoint1[27261] = {X 38.0725, Y 40.8340, Z -2.1667, A 0.000, B 0.000, C 0.000 }
gfCNCPoint1[27262] = {X 38.9100, Y 40.3375, Z -2.1667, A 0.000, B 0.000, C 0.000 }
gfCNCPoint1[27263] = {X 39.0318, Y 40.2161, Z -2.1667, A 0.000, B 0.000, C 0.000 }
gfCNCPoint1[27264] = {X 39.6099, Y 38.8458, Z -2.1667, A 0.000, B 0.000, C 0.000 }
gfCNCPoint1[27265] = {X 40.1406, Y 37.4565, Z -2.1667, A 0.000, B 0.000, C 0.000 }
gfCNCPoint1[27266] = {X 43.7124, Y 27.8657, Z -2.1667, A 0.000, B 0.000, C 0.000 }
gfCNCPoint1[27267] = {X 39.9639, Y 26.4697, Z -2.1667, A 0.000, B 0.000, C 0.000 }
gfCNCPoint1[27268] = {X 43.7874, Y 27.8937, Z -2.1667, A 0.000, B 0.000, C 0.000 }
gfCNCPoint1[27269] = {X 48.4687, Y 15.3238, Z -2.1667, A 0.000, B 0.000, C 0.000 }
gfCNCPoint1[27270] = {X 48.0765, Y 14.6072, Z -2.1667, A 0.000, B 0.000, C 0.000 }
gfCNCPoint1[27271] = {X 47.8320, Y 13.8279, Z -2.1667, A 0.000, B 0.000, C 0.000 }
gfCNCPoint1[27272] = {X 47.7444, Y 13.0158, Z -2.1667, A 0.000, B 0.000, C 0.000 }
gfCNCPoint1[27273] = {X 47.7442, Y 12.1868, Z -2.1667, A 0.000, B 0.000, C 0.000 }
gfCNCPoint1[27274] = {X 47.8485, Y 11.2611, Z -2.1667, A 0.000, B 0.000, C 0.000 }
gfCNCPoint1[27275] = {X 48.1562, Y 10.3819, Z -2.1667, A 0.000, B 0.000, C 0.000 }
gfCNCPoint1[27276] = {X 48.6518, Y 9.5931, Z -2.1667, A 0.000, B 0.000, C 0.000 }
gfCNCPoint1[27277] = {X 49.3105, Y 8.9344, Z -2.1667, A 0.000, B 0.000, C 0.000 }
gfCNCPoint1[27278] = {X 50.0993, Y 8.4388, Z -2.1667, A 0.000, B 0.000, C 0.000 }
gfCNCPoint1[27279] = {X 50.9785, Y 8.1311, Z -2.1667, A 0.000, B 0.000, C 0.000 }
gfCNCPoint1[27280] = {X 51.9042, Y 8.0268, Z -2.1667, A 0.000, B 0.000, C 0.000 }
gfCNCPoint1[27281] = {X 59.6221, Y 8.0268, Z -2.1667, A 0.000, B 0.000, C 0.000 }
gfCNCPoint1[27282] = {X 60.5478, Y 8.1311, Z -2.1667, A 0.000, B 0.000, C 0.000 }
gfCNCPoint1[27283] = {X 61.4271, Y 8.4388, Z -2.1667, A 0.000, B 0.000, C 0.000 }
gfCNCPoint1[27284] = {X 62.2158, Y 8.9344, Z -2.1667, A 0.000, B 0.000, C 0.000 }
gfCNCPoint1[27285] = {X 62.8745, Y 9.5931, Z -2.1667, A 0.000, B 0.000, C 0.000 }
gfCNCPoint1[27286] = {X 63.3702, Y 10.3819, Z -2.1667, A 0.000, B 0.000, C 0.000 }
gfCNCPoint1[27287] = {X 63.6778, Y 11.2611, Z -2.1667, A 0.000, B 0.000, C 0.000 }
gfCNCPoint1[27288] = {X 63.7821, Y 12.1868, Z -2.1667, A 0.000, B 0.000, C 0.000 }
gfCNCPoint1[27289] = {X 63.7821, Y 12.9781, Z -2.1667, A 0.000, B 0.000, C 0.000 }
gfCNCPoint1[27290] = {X 63.6960, Y 13.8204, Z -2.1667, A 0.000, B 0.000, C 0.000 }
gfCNCPoint1[27291] = {X 63.4410, Y 14.6277, Z -2.1667, A 0.000, B 0.000, C 0.000 }
gfCNCPoint1[27292] = {X 63.0280, Y 15.3667, Z -2.1667, A 0.000, B 0.000, C 0.000 }
gfCNCPoint1[27293] = {X 63.3201, Y 16.1303, Z -2.1667, A 0.000, B 0.000, C 0.000 }
gfCNCPoint1[27294] = {X 65.8843, Y 22.9436, Z -2.1667, A 0.000, B 0.000, C 0.000 }
gfCNCPoint1[27295] = {X 72.0593, Y 39.5578, Z -2.1667, A 0.000, B 0.000, C 0.000 }
gfCNCPoint1[27296] = {X 72.3893, Y 40.3878, Z -2.1667, A 0.000, B 0.000, C 0.000 }
gfCNCPoint1[27297] = {X 73.2205, Y 40.8659, Z -2.1667, A 0.000, B 0.000, C 0.000 }
gfCNCPoint1[27298] = {X 73.9202, Y 41.5217, Z -2.1667, A 0.000, B 0.000, C 0.000 }
gfCNCPoint1[27299] = {X 74.4511, Y 42.3202, Z -2.1667, A 0.000, B 0.000, C 0.000 }
gfCNCPoint1[27300] = {X 74.7850, Y 43.2191, Z -2.1667, A 0.000, B 0.000, C 0.000 }
gfCNCPoint1[27301] = {X 74.9043, Y 44.1706, Z -2.1667, A 0.000, B 0.000, C 0.000 }
gfCNCPoint1[27302] = {X 74.9045, Y 45.0000, Z -2.1667, A 0.000, B 0.000, C 0.000 }
gfCNCPoint1[27303] = {X 74.8002, Y 45.9257, Z -2.1667, A 0.000, B 0.000, C 0.000 }
gfCNCPoint1[27304] = {X 74.4925, Y 46.8050, Z -2.1667, A 0.000, B 0.000, C 0.000 }
gfCNCPoint1[27305] = {X 73.9969, Y 47.5937, Z -2.1667, A 0.000, B 0.000, C 0.000 }
gfCNCPoint1[27306] = {X 73.3382, Y 48.2524, Z -2.1667, A 0.000, B 0.000, C 0.000 }
gfCNCPoint1[27307] = {X 72.5494, Y 48.7480, Z -2.1667, A 0.000, B 0.000, C 0.000 }
gfCNCPoint1[27308] = {X 71.6701, Y 49.0557, Z -2.1667, A 0.000, B 0.000, C 0.000 }
gfCNCPoint1[27309] = {X 70.7445, Y 49.1600, Z -2.1667, A 0.000, B 0.000, C 0.000 }
gfCNCPoint1[27310] = {X 64.1851, Y 49.1600, Z -2.1667, A 0.000, B 0.000, C 0.000 }
gfCNCPoint1[27311] = {X 63.2594, Y 49.0557, Z -2.1667, A 0.000, B 0.000, C 0.000 }
gfCNCPoint1[27312] = {X 62.3802, Y 48.7480, Z -2.1667, A 0.000, B 0.000, C 0.000 }
gfCNCPoint1[27313] = {X 61.5914, Y 48.2524, Z -2.1667, A 0.000, B 0.000, C 0.000 }
gfCNCPoint1[27314] = {X 60.9327, Y 47.5937, Z -2.1667, A 0.000, B 0.000, C 0.000 }
gfCNCPoint1[27315] = {X 60.4371, Y 46.8050, Z -2.1667, A 0.000, B 0.000, C 0.000 }
gfCNCPoint1[27316] = {X 60.1294, Y 45.9257, Z -2.1667, A 0.000, B 0.000, C 0.000 }
gfCNCPoint1[27317] = {X 60.0251, Y 45.0000, Z -2.1667, A 0.000, B 0.000, C 0.000 }
gfCNCPoint1[27318] = {X 60.0251, Y 44.2086, Z -2.1667, A 0.000, B 0.000, C 0.000 }
gfCNCPoint1[27319] = {X 60.1144, Y 43.3551, Z -2.1667, A 0.000, B 0.000, C 0.000 }
gfCNCPoint1[27320] = {X 60.3769, Y 42.5382, Z -2.1667, A 0.000, B 0.000, C 0.000 }
gfCNCPoint1[27321] = {X 60.8014, Y 41.7925, Z -2.1667, A 0.000, B 0.000, C 0.000 }
gfCNCPoint1[27322] = {X 60.1192, Y 39.9292, Z -2.1667, A 0.000, B 0.000, C 0.000 }
gfCNCPoint1[27323] = {X 51.9653, Y 39.9292, Z -2.1667, A 0.000, B 0.000, C 0.000 }
gfCNCPoint1[27324] = {X 51.1569, Y 42.1007, Z -2.1667, A 0.000, B 0.000, C 0.000 }
gfCNCPoint1[27325] = {X 51.1990, Y 42.1699, Z -2.1667, A 0.000, B 0.000, C 0.000 }
gfCNCPoint1[27326] = {X 51.4888, Y 42.8045, Z -2.1667, A 0.000, B 0.000, C 0.000 }
gfCNCPoint1[27327] = {X 51.6684, Y 43.4787, Z -2.1667, A 0.000, B 0.000, C 0.000 }
gfCNCPoint1[27328] = {X 51.7328, Y 44.1733, Z -2.1667, A 0.000, B 0.000, C 0.000 }
gfCNCPoint1[27329] = {X 51.7329, Y 45.0000, Z -2.1667, A 0.000, B 0.000, C 0.000 }
gfCNCPoint1[27330] = {X 51.6286, Y 45.9257, Z -2.1667, A 0.000, B 0.000, C 0.000 }
gfCNCPoint1[27331] = {X 51.3210, Y 46.8050, Z -2.1667, A 0.000, B 0.000, C 0.000 }
gfCNCPoint1[27332] = {X 50.8253, Y 47.5937, Z -2.1667, A 0.000, B 0.000, C 0.000 }
gfCNCPoint1[27333] = {X 50.1666, Y 48.2524, Z -2.1667, A 0.000, B 0.000, C 0.000 }
gfCNCPoint1[27334] = {X 49.3779, Y 48.7480, Z -2.1667, A 0.000, B 0.000, C 0.000 }
gfCNCPoint1[27335] = {X 48.4986, Y 49.0557, Z -2.1667, A 0.000, B 0.000, C 0.000 }
gfCNCPoint1[27336] = {X 47.5729, Y 49.1600, Z -2.1667, A 0.000, B 0.000, C 0.000 }
gfCNCPoint1[27337] = {X 40.6393, Y 49.1600, Z -2.1667, A 0.000, B 0.000, C 0.000 }
gfCNCPoint1[27338] = {X 39.7136, Y 49.0557, Z -2.1667, A 0.000, B 0.000, C 0.000 }
gfCNCPoint1[27339] = {X 38.8343, Y 48.7480, Z -2.1667, A 0.000, B 0.000, C 0.000 }
gfCNCPoint1[27340] = {X 38.0456, Y 48.2524, Z -2.1667, A 0.000, B 0.000, C 0.000 }
gfCNCPoint1[27341] = {X 37.3869, Y 47.5937, Z -2.1667, A 0.000, B 0.000, C 0.000 }
gfCNCPoint1[27342] = {X 36.8913, Y 46.8050, Z -2.1667, A 0.000, B 0.000, C 0.000 }
gfCNCPoint1[27343] = {X 36.5836, Y 45.9257, Z -2.1667, A 0.000, B 0.000, C 0.000 }
gfCNCPoint1[27344] = {X 36.4793, Y 45.0000, Z -2.1667, A 0.000, B 0.000, C 0.000 }
gfCNCPoint1[27345] = {X 36.4793, Y 44.2086, Z -2.1667, A 0.000, B 0.000, C 0.000 }
gfCNCPoint1[27346] = {X 36.5897, Y 43.2569, Z -2.1667, A 0.000, B 0.000, C 0.000 }
gfCNCPoint1[27347] = {X 36.9149, Y 42.3556, Z -2.1667, A 0.000, B 0.000, C 0.000 }
gfCNCPoint1[27348] = {X 37.4376, Y 41.5527, Z -2.1667, A 0.000, B 0.000, C 0.000 }
gfCNCPoint1[27349] = {X 38.1302, Y 40.8906, Z -2.1667, A 0.000, B 0.000, C 0.000 }
gfCNCPoint1[27350] = {X 38.9560, Y 40.4046, Z -2.1667, A 0.000, B 0.000, C 0.000 }
gfCNCPoint1[27351] = {X 39.0989, Y 40.2622, Z -2.1667, A 0.000, B 0.000, C 0.000 }
gfCNCPoint1[27352] = {X 39.6813, Y 38.8826, Z -2.1667, A 0.000, B 0.000, C 0.000 }
gfCNCPoint1[27353] = {X 40.2158, Y 37.4838, Z -2.1667, A 0.000, B 0.000, C 0.000 }
gfCNCPoint1[27354] = {X 43.7874, Y 27.8937, Z -2.1667, A 0.000, B 0.000, C 0.000 }
gfCNCPoint1[27355] = {X 40.0389, Y 26.4977, Z -2.1667, A 0.000, B 0.000, C 0.000 }
gfCNCPoint1[27356] = {X 40.0389, Y 26.4976, Z -2.1667, A 0.000, B 0.000, C 0.000 }
gfCNCPoint1[27357] = {X 43.8623, Y 27.9216, Z -2.1667, A 0.000, B 0.000, C 0.000 }
gfCNCPoint1[27358] = {X 48.5582, Y 15.3126, Z -2.1667, A 0.000, B 0.000, C 0.000 }
gfCNCPoint1[27359] = {X 48.1610, Y 14.6012, Z -2.1667, A 0.000, B 0.000, C 0.000 }
gfCNCPoint1[27360] = {X 47.9131, Y 13.8250, Z -2.1667, A 0.000, B 0.000, C 0.000 }
gfCNCPoint1[27361] = {X 47.8244, Y 13.0151, Z -2.1667, A 0.000, B 0.000, C 0.000 }
gfCNCPoint1[27362] = {X 47.8242, Y 12.1868, Z -2.1667, A 0.000, B 0.000, C 0.000 }
gfCNCPoint1[27363] = {X 47.9265, Y 11.2789, Z -2.1667, A 0.000, B 0.000, C 0.000 }
gfCNCPoint1[27364] = {X 48.2283, Y 10.4166, Z -2.1667, A 0.000, B 0.000, C 0.000 }
gfCNCPoint1[27365] = {X 48.7144, Y 9.6430, Z -2.1667, A 0.000, B 0.000, C 0.000 }
gfCNCPoint1[27366] = {X 49.3604, Y 8.9969, Z -2.1667, A 0.000, B 0.000, C 0.000 }
gfCNCPoint1[27367] = {X 50.1340, Y 8.5109, Z -2.1667, A 0.000, B 0.000, C 0.000 }
gfCNCPoint1[27368] = {X 50.9963, Y 8.2091, Z -2.1667, A 0.000, B 0.000, C 0.000 }
gfCNCPoint1[27369] = {X 51.9042, Y 8.1068, Z -2.1667, A 0.000, B 0.000, C 0.000 }
gfCNCPoint1[27370] = {X 59.6221, Y 8.1068, Z -2.1667, A 0.000, B 0.000, C 0.000 }
gfCNCPoint1[27371] = {X 60.5300, Y 8.2091, Z -2.1667, A 0.000, B 0.000, C 0.000 }
gfCNCPoint1[27372] = {X 61.3924, Y 8.5109, Z -2.1667, A 0.000, B 0.000, C 0.000 }
gfCNCPoint1[27373] = {X 62.1660, Y 8.9969, Z -2.1667, A 0.000, B 0.000, C 0.000 }
gfCNCPoint1[27374] = {X 62.8120, Y 9.6430, Z -2.1667, A 0.000, B 0.000, C 0.000 }
gfCNCPoint1[27375] = {X 63.2981, Y 10.4166, Z -2.1667, A 0.000, B 0.000, C 0.000 }
gfCNCPoint1[27376] = {X 63.5998, Y 11.2789, Z -2.1667, A 0.000, B 0.000, C 0.000 }
gfCNCPoint1[27377] = {X 63.7021, Y 12.1868, Z -2.1667, A 0.000, B 0.000, C 0.000 }
gfCNCPoint1[27378] = {X 63.7021, Y 12.9781, Z -2.1667, A 0.000, B 0.000, C 0.000 }
gfCNCPoint1[27379] = {X 63.6147, Y 13.8180, Z -2.1667, A 0.000, B 0.000, C 0.000 }
gfCNCPoint1[27380] = {X 63.3563, Y 14.6219, Z -2.1667, A 0.000, B 0.000, C 0.000 }
gfCNCPoint1[27381] = {X 62.9379, Y 15.3554, Z -2.1667, A 0.000, B 0.000, C 0.000 }
gfCNCPoint1[27382] = {X 63.2453, Y 16.1586, Z -2.1667, A 0.000, B 0.000, C 0.000 }
gfCNCPoint1[27383] = {X 65.8094, Y 22.9716, Z -2.1667, A 0.000, B 0.000, C 0.000 }
gfCNCPoint1[27384] = {X 71.9847, Y 39.5865, Z -2.1667, A 0.000, B 0.000, C 0.000 }
gfCNCPoint1[27385] = {X 72.3273, Y 40.4483, Z -2.1667, A 0.000, B 0.000, C 0.000 }
gfCNCPoint1[27386] = {X 73.1516, Y 40.9146, Z -2.1667, A 0.000, B 0.000, C 0.000 }
gfCNCPoint1[27387] = {X 73.8463, Y 41.5583, Z -2.1667, A 0.000, B 0.000, C 0.000 }
gfCNCPoint1[27388] = {X 74.3738, Y 42.3448, Z -2.1667, A 0.000, B 0.000, C 0.000 }
gfCNCPoint1[27389] = {X 74.7057, Y 43.2318, Z -2.1667, A 0.000, B 0.000, C 0.000 }
gfCNCPoint1[27390] = {X 74.8243, Y 44.1714, Z -2.1667, A 0.000, B 0.000, C 0.000 }
gfCNCPoint1[27391] = {X 74.8245, Y 45.0000, Z -2.1667, A 0.000, B 0.000, C 0.000 }
gfCNCPoint1[27392] = {X 74.7222, Y 45.9079, Z -2.1667, A 0.000, B 0.000, C 0.000 }
gfCNCPoint1[27393] = {X 74.4204, Y 46.7702, Z -2.1667, A 0.000, B 0.000, C 0.000 }
gfCNCPoint1[27394] = {X 73.9343, Y 47.5438, Z -2.1667, A 0.000, B 0.000, C 0.000 }
gfCNCPoint1[27395] = {X 73.2883, Y 48.1899, Z -2.1667, A 0.000, B 0.000, C 0.000 }
gfCNCPoint1[27396] = {X 72.5147, Y 48.6760, Z -2.1667, A 0.000, B 0.000, C 0.000 }
gfCNCPoint1[27397] = {X 71.6523, Y 48.9777, Z -2.1667, A 0.000, B 0.000, C 0.000 }
gfCNCPoint1[27398] = {X 70.7445, Y 49.0800, Z -2.1667, A 0.000, B 0.000, C 0.000 }
gfCNCPoint1[27399] = {X 64.1851, Y 49.0800, Z -2.1667, A 0.000, B 0.000, C 0.000 }
gfCNCPoint1[27400] = {X 63.2772, Y 48.9777, Z -2.1667, A 0.000, B 0.000, C 0.000 }
gfCNCPoint1[27401] = {X 62.4149, Y 48.6760, Z -2.1667, A 0.000, B 0.000, C 0.000 }
gfCNCPoint1[27402] = {X 61.6413, Y 48.1899, Z -2.1667, A 0.000, B 0.000, C 0.000 }
gfCNCPoint1[27403] = {X 60.9953, Y 47.5438, Z -2.1667, A 0.000, B 0.000, C 0.000 }
gfCNCPoint1[27404] = {X 60.5092, Y 46.7702, Z -2.1667, A 0.000, B 0.000, C 0.000 }
gfCNCPoint1[27405] = {X 60.2074, Y 45.9079, Z -2.1667, A 0.000, B 0.000, C 0.000 }
gfCNCPoint1[27406] = {X 60.1051, Y 45.0000, Z -2.1667, A 0.000, B 0.000, C 0.000 }
gfCNCPoint1[27407] = {X 60.1051, Y 44.2086, Z -2.1667, A 0.000, B 0.000, C 0.000 }
gfCNCPoint1[27408] = {X 60.1956, Y 43.3579, Z -2.1667, A 0.000, B 0.000, C 0.000 }
gfCNCPoint1[27409] = {X 60.4615, Y 42.5447, Z -2.1667, A 0.000, B 0.000, C 0.000 }
gfCNCPoint1[27410] = {X 60.8911, Y 41.8049, Z -2.1667, A 0.000, B 0.000, C 0.000 }
gfCNCPoint1[27411] = {X 60.1751, Y 39.8492, Z -2.1667, A 0.000, B 0.000, C 0.000 }
gfCNCPoint1[27412] = {X 51.9097, Y 39.8492, Z -2.1667, A 0.000, B 0.000, C 0.000 }
gfCNCPoint1[27413] = {X 51.0684, Y 42.1091, Z -2.1667, A 0.000, B 0.000, C 0.000 }
gfCNCPoint1[27414] = {X 51.1306, Y 42.2115, Z -2.1667, A 0.000, B 0.000, C 0.000 }
gfCNCPoint1[27415] = {X 51.4141, Y 42.8332, Z -2.1667, A 0.000, B 0.000, C 0.000 }
gfCNCPoint1[27416] = {X 51.5898, Y 43.4936, Z -2.1667, A 0.000, B 0.000, C 0.000 }
gfCNCPoint1[27417] = {X 51.6528, Y 44.1740, Z -2.1667, A 0.000, B 0.000, C 0.000 }
gfCNCPoint1[27418] = {X 51.6529, Y 45.0000, Z -2.1667, A 0.000, B 0.000, C 0.000 }
gfCNCPoint1[27419] = {X 51.5506, Y 45.9079, Z -2.1667, A 0.000, B 0.000, C 0.000 }
gfCNCPoint1[27420] = {X 51.2489, Y 46.7702, Z -2.1667, A 0.000, B 0.000, C 0.000 }
gfCNCPoint1[27421] = {X 50.7628, Y 47.5438, Z -2.1667, A 0.000, B 0.000, C 0.000 }
gfCNCPoint1[27422] = {X 50.1168, Y 48.1899, Z -2.1667, A 0.000, B 0.000, C 0.000 }
gfCNCPoint1[27423] = {X 49.3432, Y 48.6760, Z -2.1667, A 0.000, B 0.000, C 0.000 }
gfCNCPoint1[27424] = {X 48.4808, Y 48.9777, Z -2.1667, A 0.000, B 0.000, C 0.000 }
gfCNCPoint1[27425] = {X 47.5729, Y 49.0800, Z -2.1667, A 0.000, B 0.000, C 0.000 }
gfCNCPoint1[27426] = {X 40.6393, Y 49.0800, Z -2.1667, A 0.000, B 0.000, C 0.000 }
gfCNCPoint1[27427] = {X 39.7314, Y 48.9777, Z -2.1667, A 0.000, B 0.000, C 0.000 }
gfCNCPoint1[27428] = {X 38.8691, Y 48.6760, Z -2.1667, A 0.000, B 0.000, C 0.000 }
gfCNCPoint1[27429] = {X 38.0955, Y 48.1899, Z -2.1667, A 0.000, B 0.000, C 0.000 }
gfCNCPoint1[27430] = {X 37.4494, Y 47.5438, Z -2.1667, A 0.000, B 0.000, C 0.000 }
gfCNCPoint1[27431] = {X 36.9633, Y 46.7702, Z -2.1667, A 0.000, B 0.000, C 0.000 }
gfCNCPoint1[27432] = {X 36.6616, Y 45.9079, Z -2.1667, A 0.000, B 0.000, C 0.000 }
gfCNCPoint1[27433] = {X 36.5593, Y 45.0000, Z -2.1667, A 0.000, B 0.000, C 0.000 }
gfCNCPoint1[27434] = {X 36.5593, Y 44.2087, Z -2.1667, A 0.000, B 0.000, C 0.000 }
gfCNCPoint1[27435] = {X 36.6682, Y 43.2723, Z -2.1667, A 0.000, B 0.000, C 0.000 }
gfCNCPoint1[27436] = {X 36.9891, Y 42.3860, Z -2.1667, A 0.000, B 0.000, C 0.000 }
gfCNCPoint1[27437] = {X 37.5049, Y 41.5969, Z -2.1667, A 0.000, B 0.000, C 0.000 }
gfCNCPoint1[27438] = {X 38.1879, Y 40.9473, Z -2.1667, A 0.000, B 0.000, C 0.000 }
gfCNCPoint1[27439] = {X 39.0018, Y 40.4718, Z -2.1667, A 0.000, B 0.000, C 0.000 }
gfCNCPoint1[27440] = {X 39.1660, Y 40.3083, Z -2.1667, A 0.000, B 0.000, C 0.000 }
gfCNCPoint1[27441] = {X 39.7528, Y 38.9194, Z -2.1667, A 0.000, B 0.000, C 0.000 }
gfCNCPoint1[27442] = {X 40.2910, Y 37.5110, Z -2.1667, A 0.000, B 0.000, C 0.000 }
gfCNCPoint1[27443] = {X 43.8623, Y 27.9216, Z -2.1667, A 0.000, B 0.000, C 0.000 }
gfCNCPoint1[27444] = {X 40.1139, Y 26.5256, Z -2.1667, A 0.000, B 0.000, C 0.000 }
gfCNCPoint1[27445] = {X 43.9373, Y 27.9495, Z -2.1667, A 0.000, B 0.000, C 0.000 }
gfCNCPoint1[27446] = {X 48.6479, Y 15.3010, Z -2.1667, A 0.000, B 0.000, C 0.000 }
gfCNCPoint1[27447] = {X 48.2407, Y 14.5838, Z -2.1667, A 0.000, B 0.000, C 0.000 }
gfCNCPoint1[27448] = {X 47.9892, Y 13.7983, Z -2.1667, A 0.000, B 0.000, C 0.000 }
gfCNCPoint1[27449] = {X 47.9042, Y 12.9779, Z -2.1667, A 0.000, B 0.000, C 0.000 }
gfCNCPoint1[27450] = {X 47.9042, Y 12.1868, Z -2.1667, A 0.000, B 0.000, C 0.000 }
gfCNCPoint1[27451] = {X 48.0045, Y 11.2967, Z -2.1667, A 0.000, B 0.000, C 0.000 }
gfCNCPoint1[27452] = {X 48.3003, Y 10.4513, Z -2.1667, A 0.000, B 0.000, C 0.000 }
gfCNCPoint1[27453] = {X 48.7769, Y 9.6929, Z -2.1667, A 0.000, B 0.000, C 0.000 }
gfCNCPoint1[27454] = {X 49.4103, Y 9.0595, Z -2.1667, A 0.000, B 0.000, C 0.000 }
gfCNCPoint1[27455] = {X 50.1687, Y 8.5829, Z -2.1667, A 0.000, B 0.000, C 0.000 }
gfCNCPoint1[27456] = {X 51.0141, Y 8.2871, Z -2.1667, A 0.000, B 0.000, C 0.000 }
gfCNCPoint1[27457] = {X 51.9042, Y 8.1868, Z -2.1667, A 0.000, B 0.000, C 0.000 }
gfCNCPoint1[27458] = {X 59.6221, Y 8.1868, Z -2.1667, A 0.000, B 0.000, C 0.000 }
gfCNCPoint1[27459] = {X 60.5122, Y 8.2871, Z -2.1667, A 0.000, B 0.000, C 0.000 }
gfCNCPoint1[27460] = {X 61.3577, Y 8.5829, Z -2.1667, A 0.000, B 0.000, C 0.000 }
gfCNCPoint1[27461] = {X 62.1161, Y 9.0595, Z -2.1667, A 0.000, B 0.000, C 0.000 }
gfCNCPoint1[27462] = {X 62.7495, Y 9.6929, Z -2.1667, A 0.000, B 0.000, C 0.000 }
gfCNCPoint1[27463] = {X 63.2260, Y 10.4513, Z -2.1667, A 0.000, B 0.000, C 0.000 }
gfCNCPoint1[27464] = {X 63.5218, Y 11.2967, Z -2.1667, A 0.000, B 0.000, C 0.000 }
gfCNCPoint1[27465] = {X 63.6221, Y 12.1868, Z -2.1667, A 0.000, B 0.000, C 0.000 }
gfCNCPoint1[27466] = {X 63.6219, Y 13.0192, Z -2.1667, A 0.000, B 0.000, C 0.000 }
gfCNCPoint1[27467] = {X 63.5276, Y 13.8423, Z -2.1667, A 0.000, B 0.000, C 0.000 }
gfCNCPoint1[27468] = {X 63.2658, Y 14.6283, Z -2.1667, A 0.000, B 0.000, C 0.000 }
gfCNCPoint1[27469] = {X 62.8477, Y 15.3435, Z -2.1667, A 0.000, B 0.000, C 0.000 }
gfCNCPoint1[27470] = {X 63.1705, Y 16.1870, Z -2.1667, A 0.000, B 0.000, C 0.000 }
gfCNCPoint1[27471] = {X 65.7344, Y 22.9996, Z -2.1667, A 0.000, B 0.000, C 0.000 }
gfCNCPoint1[27472] = {X 71.9100, Y 39.6152, Z -2.1667, A 0.000, B 0.000, C 0.000 }
gfCNCPoint1[27473] = {X 72.2607, Y 40.4974, Z -2.1667, A 0.000, B 0.000, C 0.000 }
gfCNCPoint1[27474] = {X 72.2771, Y 40.5141, Z -2.1667, A 0.000, B 0.000, C 0.000 }
gfCNCPoint1[27475] = {X 72.3436, Y 40.5424, Z -2.1667, A 0.000, B 0.000, C 0.000 }
gfCNCPoint1[27476] = {X 72.4097, Y 40.5719, Z -2.1667, A 0.000, B 0.000, C 0.000 }
gfCNCPoint1[27477] = {X 73.1895, Y 41.0431, Z -2.1667, A 0.000, B 0.000, C 0.000 }
gfCNCPoint1[27478] = {X 73.8425, Y 41.6786, Z -2.1667, A 0.000, B 0.000, C 0.000 }
gfCNCPoint1[27479] = {X 74.3348, Y 42.4454, Z -2.1667, A 0.000, B 0.000, C 0.000 }
gfCNCPoint1[27480] = {X 74.6407, Y 43.3037, Z -2.1667, A 0.000, B 0.000, C 0.000 }
gfCNCPoint1[27481] = {X 74.7445, Y 44.2089, Z -2.1667, A 0.000, B 0.000, C 0.000 }
gfCNCPoint1[27482] = {X 74.7445, Y 45.0000, Z -2.1667, A 0.000, B 0.000, C 0.000 }
gfCNCPoint1[27483] = {X 74.6442, Y 45.8901, Z -2.1667, A 0.000, B 0.000, C 0.000 }
gfCNCPoint1[27484] = {X 74.3483, Y 46.7355, Z -2.1667, A 0.000, B 0.000, C 0.000 }
gfCNCPoint1[27485] = {X 73.8718, Y 47.4940, Z -2.1667, A 0.000, B 0.000, C 0.000 }
gfCNCPoint1[27486] = {X 73.2384, Y 48.1273, Z -2.1667, A 0.000, B 0.000, C 0.000 }
gfCNCPoint1[27487] = {X 72.4800, Y 48.6039, Z -2.1667, A 0.000, B 0.000, C 0.000 }
gfCNCPoint1[27488] = {X 71.6345, Y 48.8997, Z -2.1667, A 0.000, B 0.000, C 0.000 }
gfCNCPoint1[27489] = {X 70.7445, Y 49.0000, Z -2.1667, A 0.000, B 0.000, C 0.000 }
gfCNCPoint1[27490] = {X 64.1851, Y 49.0000, Z -2.1667, A 0.000, B 0.000, C 0.000 }
gfCNCPoint1[27491] = {X 63.2951, Y 48.8997, Z -2.1667, A 0.000, B 0.000, C 0.000 }
gfCNCPoint1[27492] = {X 62.4496, Y 48.6039, Z -2.1667, A 0.000, B 0.000, C 0.000 }
gfCNCPoint1[27493] = {X 61.6912, Y 48.1273, Z -2.1667, A 0.000, B 0.000, C 0.000 }
gfCNCPoint1[27494] = {X 61.0578, Y 47.4940, Z -2.1667, A 0.000, B 0.000, C 0.000 }
gfCNCPoint1[27495] = {X 60.5813, Y 46.7355, Z -2.1667, A 0.000, B 0.000, C 0.000 }
gfCNCPoint1[27496] = {X 60.2854, Y 45.8901, Z -2.1667, A 0.000, B 0.000, C 0.000 }
gfCNCPoint1[27497] = {X 60.1851, Y 45.0000, Z -2.1667, A 0.000, B 0.000, C 0.000 }
gfCNCPoint1[27498] = {X 60.1855, Y 44.1538, Z -2.1667, A 0.000, B 0.000, C 0.000 }
gfCNCPoint1[27499] = {X 60.2746, Y 43.3674, Z -2.1667, A 0.000, B 0.000, C 0.000 }
gfCNCPoint1[27500] = {X 60.5168, Y 42.6140, Z -2.1667, A 0.000, B 0.000, C 0.000 }
gfCNCPoint1[27501] = {X 60.9025, Y 41.9231, Z -2.1667, A 0.000, B 0.000, C 0.000 }
gfCNCPoint1[27502] = {X 60.9811, Y 41.8181, Z -2.1667, A 0.000, B 0.000, C 0.000 }
gfCNCPoint1[27503] = {X 60.2310, Y 39.7692, Z -2.1667, A 0.000, B 0.000, C 0.000 }
gfCNCPoint1[27504] = {X 51.8419, Y 39.7692, Z -2.1667, A 0.000, B 0.000, C 0.000 }
gfCNCPoint1[27505] = {X 51.8419, Y 39.8021, Z -2.1667, A 0.000, B 0.000, C 0.000 }
gfCNCPoint1[27506] = {X 50.9799, Y 42.1175, Z -2.1667, A 0.000, B 0.000, C 0.000 }
gfCNCPoint1[27507] = {X 51.0720, Y 42.2706, Z -2.1667, A 0.000, B 0.000, C 0.000 }
gfCNCPoint1[27508] = {X 51.3476, Y 42.8854, Z -2.1667, A 0.000, B 0.000, C 0.000 }
gfCNCPoint1[27509] = {X 51.5162, Y 43.5376, Z -2.1667, A 0.000, B 0.000, C 0.000 }
gfCNCPoint1[27510] = {X 51.5729, Y 44.2089, Z -2.1667, A 0.000, B 0.000, C 0.000 }
gfCNCPoint1[27511] = {X 51.5729, Y 45.0000, Z -2.1667, A 0.000, B 0.000, C 0.000 }
gfCNCPoint1[27512] = {X 51.4726, Y 45.8901, Z -2.1667, A 0.000, B 0.000, C 0.000 }
gfCNCPoint1[27513] = {X 51.1768, Y 46.7355, Z -2.1667, A 0.000, B 0.000, C 0.000 }
gfCNCPoint1[27514] = {X 50.7003, Y 47.4940, Z -2.1667, A 0.000, B 0.000, C 0.000 }
gfCNCPoint1[27515] = {X 50.0669, Y 48.1273, Z -2.1667, A 0.000, B 0.000, C 0.000 }
gfCNCPoint1[27516] = {X 49.3085, Y 48.6039, Z -2.1667, A 0.000, B 0.000, C 0.000 }
gfCNCPoint1[27517] = {X 48.4630, Y 48.8997, Z -2.1667, A 0.000, B 0.000, C 0.000 }
gfCNCPoint1[27518] = {X 47.5729, Y 49.0000, Z -2.1667, A 0.000, B 0.000, C 0.000 }
gfCNCPoint1[27519] = {X 40.6393, Y 49.0000, Z -2.1667, A 0.000, B 0.000, C 0.000 }
gfCNCPoint1[27520] = {X 39.7492, Y 48.8997, Z -2.1667, A 0.000, B 0.000, C 0.000 }
gfCNCPoint1[27521] = {X 38.9038, Y 48.6039, Z -2.1667, A 0.000, B 0.000, C 0.000 }
gfCNCPoint1[27522] = {X 38.1453, Y 48.1273, Z -2.1667, A 0.000, B 0.000, C 0.000 }
gfCNCPoint1[27523] = {X 37.5120, Y 47.4940, Z -2.1667, A 0.000, B 0.000, C 0.000 }
gfCNCPoint1[27524] = {X 37.0354, Y 46.7355, Z -2.1667, A 0.000, B 0.000, C 0.000 }
gfCNCPoint1[27525] = {X 36.7396, Y 45.8901, Z -2.1667, A 0.000, B 0.000, C 0.000 }
gfCNCPoint1[27526] = {X 36.6393, Y 45.0000, Z -2.1667, A 0.000, B 0.000, C 0.000 }
gfCNCPoint1[27527] = {X 36.6397, Y 44.1538, Z -2.1667, A 0.000, B 0.000, C 0.000 }
gfCNCPoint1[27528] = {X 36.7564, Y 43.2480, Z -2.1667, A 0.000, B 0.000, C 0.000 }
gfCNCPoint1[27529] = {X 37.0755, Y 42.3923, Z -2.1667, A 0.000, B 0.000, C 0.000 }
gfCNCPoint1[27530] = {X 37.5804, Y 41.6313, Z -2.1667, A 0.000, B 0.000, C 0.000 }
gfCNCPoint1[27531] = {X 38.2448, Y 41.0047, Z -2.1667, A 0.000, B 0.000, C 0.000 }
gfCNCPoint1[27532] = {X 39.0339, Y 40.5451, Z -2.1667, A 0.000, B 0.000, C 0.000 }
gfCNCPoint1[27533] = {X 39.0885, Y 40.5216, Z -2.1667, A 0.000, B 0.000, C 0.000 }
gfCNCPoint1[27534] = {X 39.1435, Y 40.4990, Z -2.1667, A 0.000, B 0.000, C 0.000 }
gfCNCPoint1[27535] = {X 39.1697, Y 40.4820, Z -2.1667, A 0.000, B 0.000, C 0.000 }
gfCNCPoint1[27536] = {X 39.1877, Y 40.4564, Z -2.1667, A 0.000, B 0.000, C 0.000 }
gfCNCPoint1[27537] = {X 39.2134, Y 40.3986, Z -2.1667, A 0.000, B 0.000, C 0.000 }
gfCNCPoint1[27538] = {X 39.2391, Y 40.3407, Z -2.1667, A 0.000, B 0.000, C 0.000 }
gfCNCPoint1[27539] = {X 39.8270, Y 38.9493, Z -2.1667, A 0.000, B 0.000, C 0.000 }
gfCNCPoint1[27540] = {X 40.3662, Y 37.5383, Z -2.1667, A 0.000, B 0.000, C 0.000 }
gfCNCPoint1[27541] = {X 43.9373, Y 27.9495, Z -2.1667, A 0.000, B 0.000, C 0.000 }
gfCNCPoint1[27542] = {X 40.1139, Y 26.5256, Z -2.1667, A 0.000, B 0.000, C 0.000 }
gfCNCPoint1[27543] = {X 40.1139, Y 26.5256, Z 0.8333, A 0.000, B 0.000, C 0.000 }
gfCNCPoint1[27544] = {X 40.1139, Y 26.5256, Z 11.0000, A 0.000, B 0.000, C 0.000 }
gfCNCPoint1[27545] = {X 79.0236, Y 28.5922, Z 11.0000, A 0.000, B 0.000, C 0.000 }
gfCNCPoint1[27546] = {X 79.0236, Y 28.5922, Z 0.8333, A 0.000, B 0.000, C 0.000 }
gfCNCPoint1[27547] = {X 79.0236, Y 28.5922, Z -2.1667, A 0.000, B 0.000, C 0.000 }
gfCNCPoint1[27548] = {X 83.1036, Y 28.5922, Z -2.1667, A 0.000, B 0.000, C 0.000 }
gfCNCPoint1[27549] = {X 83.1034, Y 16.2748, Z -2.1667, A 0.000, B 0.000, C 0.000 }
gfCNCPoint1[27550] = {X 82.4645, Y 15.6036, Z -2.1667, A 0.000, B 0.000, C 0.000 }
gfCNCPoint1[27551] = {X 81.9835, Y 14.8116, Z -2.1667, A 0.000, B 0.000, C 0.000 }
gfCNCPoint1[27552] = {X 81.6825, Y 13.9353, Z -2.1667, A 0.000, B 0.000, C 0.000 }
gfCNCPoint1[27553] = {X 81.5752, Y 13.0148, Z -2.1667, A 0.000, B 0.000, C 0.000 }
gfCNCPoint1[27554] = {X 81.5751, Y 12.1868, Z -2.1667, A 0.000, B 0.000, C 0.000 }
gfCNCPoint1[27555] = {X 81.6834, Y 11.2255, Z -2.1667, A 0.000, B 0.000, C 0.000 }
gfCNCPoint1[27556] = {X 82.0029, Y 10.3124, Z -2.1667, A 0.000, B 0.000, C 0.000 }
gfCNCPoint1[27557] = {X 82.5176, Y 9.4933, Z -2.1667, A 0.000, B 0.000, C 0.000 }
gfCNCPoint1[27558] = {X 83.2016, Y 8.8093, Z -2.1667, A 0.000, B 0.000, C 0.000 }
gfCNCPoint1[27559] = {X 84.0207, Y 8.2946, Z -2.1667, A 0.000, B 0.000, C 0.000 }
gfCNCPoint1[27560] = {X 84.9338, Y 7.9751, Z -2.1667, A 0.000, B 0.000, C 0.000 }
gfCNCPoint1[27561] = {X 85.8951, Y 7.8668, Z -2.1667, A 0.000, B 0.000, C 0.000 }
gfCNCPoint1[27562] = {X 94.0497, Y 7.8668, Z -2.1667, A 0.000, B 0.000, C 0.000 }
gfCNCPoint1[27563] = {X 95.0110, Y 7.9751, Z -2.1667, A 0.000, B 0.000, C 0.000 }
gfCNCPoint1[27564] = {X 95.9240, Y 8.2946, Z -2.1667, A 0.000, B 0.000, C 0.000 }
gfCNCPoint1[27565] = {X 96.7431, Y 8.8093, Z -2.1667, A 0.000, B 0.000, C 0.000 }
gfCNCPoint1[27566] = {X 97.4272, Y 9.4933, Z -2.1667, A 0.000, B 0.000, C 0.000 }
gfCNCPoint1[27567] = {X 97.9419, Y 10.3124, Z -2.1667, A 0.000, B 0.000, C 0.000 }
gfCNCPoint1[27568] = {X 98.2614, Y 11.2255, Z -2.1667, A 0.000, B 0.000, C 0.000 }
gfCNCPoint1[27569] = {X 98.3697, Y 12.1868, Z -2.1667, A 0.000, B 0.000, C 0.000 }
gfCNCPoint1[27570] = {X 98.3697, Y 12.9781, Z -2.1667, A 0.000, B 0.000, C 0.000 }
gfCNCPoint1[27571] = {X 98.2966, Y 13.7684, Z -2.1667, A 0.000, B 0.000, C 0.000 }
gfCNCPoint1[27572] = {X 98.0803, Y 14.5319, Z -2.1667, A 0.000, B 0.000, C 0.000 }
gfCNCPoint1[27573] = {X 97.7279, Y 15.2430, Z -2.1667, A 0.000, B 0.000, C 0.000 }
gfCNCPoint1[27574] = {X 101.8780, Y 25.5306, Z -2.1667, A 0.000, B 0.000, C 0.000 }
gfCNCPoint1[27575] = {X 106.0168, Y 15.2220, Z -2.1667, A 0.000, B 0.000, C 0.000 }
gfCNCPoint1[27576] = {X 105.6763, Y 14.5290, Z -2.1667, A 0.000, B 0.000, C 0.000 }
gfCNCPoint1[27577] = {X 105.4646, Y 13.7863, Z -2.1667, A 0.000, B 0.000, C 0.000 }
gfCNCPoint1[27578] = {X 105.3885, Y 13.0179, Z -2.1667, A 0.000, B 0.000, C 0.000 }
gfCNCPoint1[27579] = {X 105.3883, Y 12.1868, Z -2.1667, A 0.000, B 0.000, C 0.000 }
gfCNCPoint1[27580] = {X 105.4966, Y 11.2255, Z -2.1667, A 0.000, B 0.000, C 0.000 }
gfCNCPoint1[27581] = {X 105.8161, Y 10.3124, Z -2.1667, A 0.000, B 0.000, C 0.000 }
gfCNCPoint1[27582] = {X 106.3308, Y 9.4933, Z -2.1667, A 0.000, B 0.000, C 0.000 }
gfCNCPoint1[27583] = {X 107.0148, Y 8.8093, Z -2.1667, A 0.000, B 0.000, C 0.000 }
gfCNCPoint1[27584] = {X 107.8339, Y 8.2946, Z -2.1667, A 0.000, B 0.000, C 0.000 }
gfCNCPoint1[27585] = {X 108.7470, Y 7.9751, Z -2.1667, A 0.000, B 0.000, C 0.000 }
gfCNCPoint1[27586] = {X 109.7083, Y 7.8668, Z -2.1667, A 0.000, B 0.000, C 0.000 }
gfCNCPoint1[27587] = {X 117.7916, Y 7.8668, Z -2.1667, A 0.000, B 0.000, C 0.000 }
gfCNCPoint1[27588] = {X 118.7529, Y 7.9751, Z -2.1667, A 0.000, B 0.000, C 0.000 }
gfCNCPoint1[27589] = {X 119.6660, Y 8.2946, Z -2.1667, A 0.000, B 0.000, C 0.000 }
gfCNCPoint1[27590] = {X 120.4851, Y 8.8093, Z -2.1667, A 0.000, B 0.000, C 0.000 }
gfCNCPoint1[27591] = {X 121.1691, Y 9.4933, Z -2.1667, A 0.000, B 0.000, C 0.000 }
gfCNCPoint1[27592] = {X 121.6838, Y 10.3124, Z -2.1667, A 0.000, B 0.000, C 0.000 }
gfCNCPoint1[27593] = {X 122.0033, Y 11.2255, Z -2.1667, A 0.000, B 0.000, C 0.000 }
gfCNCPoint1[27594] = {X 122.1116, Y 12.1868, Z -2.1667, A 0.000, B 0.000, C 0.000 }
gfCNCPoint1[27595] = {X 122.1116, Y 12.9781, Z -2.1667, A 0.000, B 0.000, C 0.000 }
gfCNCPoint1[27596] = {X 122.0103, Y 13.9080, Z -2.1667, A 0.000, B 0.000, C 0.000 }
gfCNCPoint1[27597] = {X 121.7112, Y 14.7943, Z -2.1667, A 0.000, B 0.000, C 0.000 }
gfCNCPoint1[27598] = {X 121.2284, Y 15.5954, Z -2.1667, A 0.000, B 0.000, C 0.000 }
gfCNCPoint1[27599] = {X 120.5844, Y 16.2739, Z -2.1667, A 0.000, B 0.000, C 0.000 }
gfCNCPoint1[27600] = {X 120.5831, Y 40.9137, Z -2.1667, A 0.000, B 0.000, C 0.000 }
gfCNCPoint1[27601] = {X 120.6217, Y 40.9449, Z -2.1667, A 0.000, B 0.000, C 0.000 }
